iq_stStandardModuleItf.q_etDiag			:= GD.ET_Diag.Ok;
iq_stStandardModuleItf.q_udiDiagExt		:= ET_DiagExt.Disabled;
iq_stStandardModuleItf.q_sDiagExt			:= FC_EtDiagExtToString(i_etDiagExt := iq_stStandardModuleItf.q_udiDiagExt);
iq_stStandardModuleItf.q_sMsg				:= '';

iq_stStandardModuleItf.q_dwModuleType		:= TPL.ET_ModuleType.NodeModule;
iq_stStandardModuleItf.q_sModuleTypeName	:= 'NodeModule';
iq_stStandardModuleItf.q_udiModuleVersion	:= 1;	
(* End of system generated code, do not change without consulting 'Schneider Electric Automation GmbH' - otherwise you risk instability!!! *)

(* System generated code, to be changed by experienced programmers *)
IF iq_stStandardModuleItf.iq_diCMD <> 0 AND NOT iq_stStandardModuleItf.i_xEnable THEN
	iq_stStandardModuleItf.iq_diCMD := 0;
END_IF
(* End of system generated code, to be changed by experienced programmers *)

(* Application specific code *)
(* ToDo: Add your application specific code here *)
;
(* End of application specific code *)
END_ACTION

ACTION SubModules_Action:
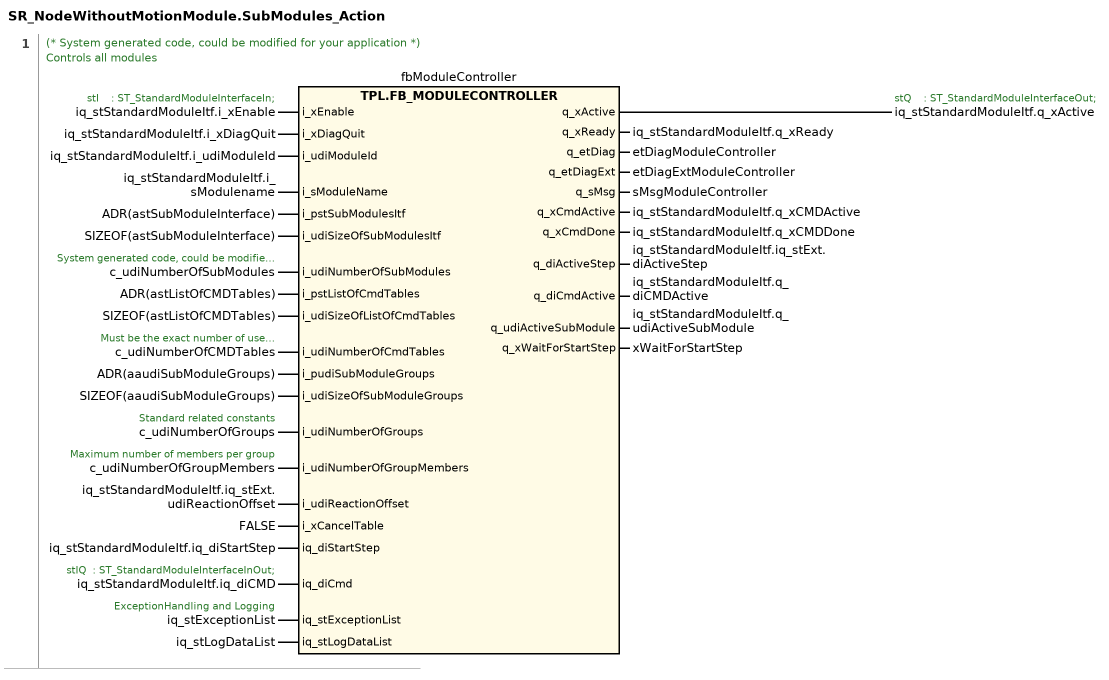
// NETWORK 1
// 					(* System generated code, could be modified for your application *)
// Controls all modules
//
//   fbModuleController: Modules related variables
//   iq_stStandardModuleItf.i_xEnable: stI : ST_StandardModuleInterfaceIn;
//   c_udiNumberOfSubModules: System generated code, could be modified for your application
//   c_udiNumberOfCMDTables: Must be the exact number of used CMDTables!
//   c_udiNumberOfGroups: Standard related constants
//   c_udiNumberOfGroupMembers: Maximum number of members per group
//   iq_stStandardModuleItf.iq_diCMD: stIQ : ST_StandardModuleInterfaceInOut;
//   iq_stExceptionList: ExceptionHandling and Logging
//   iq_stStandardModuleItf.q_xActive: stQ : ST_StandardModuleInterfaceOut;
fbModuleController(
    i_xEnable := iq_stStandardModuleItf.i_xEnable,
    i_xDiagQuit := iq_stStandardModuleItf.i_xDiagQuit,
    i_udiModuleId := iq_stStandardModuleItf.i_udiModuleId,
    i_sModuleName := iq_stStandardModuleItf.i_sModulename,
    i_pstSubModulesItf := ADR(astSubModuleInterface),
    i_udiSizeOfSubModulesItf := SIZEOF(astSubModuleInterface),
    i_udiNumberOfSubModules := c_udiNumberOfSubModules,
    i_pstListOfCmdTables := ADR(astListOfCMDTables),
    i_udiSizeOfListOfCmdTables := SIZEOF(astListOfCMDTables),
    i_udiNumberOfCmdTables := c_udiNumberOfCMDTables,
    i_pudiSubModuleGroups := ADR(aaudiSubModuleGroups),
    i_udiSizeOfSubModuleGroups := SIZEOF(aaudiSubModuleGroups),
    i_udiNumberOfGroups := c_udiNumberOfGroups,
    i_udiNumberOfGroupMembers := c_udiNumberOfGroupMembers,
    i_udiReactionOffset := iq_stStandardModuleItf.iq_stExt.udiReactionOffset,
    i_xCancelTable := FALSE,
    iq_diStartStep := iq_stStandardModuleItf.iq_diStartStep,
    iq_diCmd := iq_stStandardModuleItf.iq_diCMD,
    iq_stExceptionList := iq_stExceptionList,
    iq_stLogDataList := iq_stLogDataList,
    q_xReady => iq_stStandardModuleItf.q_xReady,
    q_etDiag => etDiagModuleController,
    q_etDiagExt => etDiagExtModuleController,
    q_sMsg => sMsgModuleController,
    q_xCmdActive => iq_stStandardModuleItf.q_xCMDActive,
    q_xCmdDone => iq_stStandardModuleItf.q_xCMDDone,
    q_diActiveStep => iq_stStandardModuleItf.iq_stExt.diActiveStep,
    q_diCmdActive => iq_stStandardModuleItf.q_diCMDActive,
    q_udiActiveSubModule => iq_stStandardModuleItf.q_udiActiveSubModule,
    q_xWaitForStartStep => xWaitForStartStep); // TPL.FB_MODULECONTROLLER
iq_stStandardModuleItf.q_xActive := fbModuleController.q_xActive;
END_ACTION

ACTION UpdateStructs:
(* System generated code, do not change without consulting 'Schneider Electric Automation GmbH' - otherwise you risk instability!!!*)
fbDetectOnlineChange(	i_xEnable	:= TRUE, 
						i_xDetect	:= TRUE, 
						q_xActive	=> xDetectOnlineChangeActive, 
						q_xReady	=> xDetectOnlineChangeReady, 
						q_etDiag	=> etDetectOnlineChangeDiag, 
						q_etDiagExt	=> etDetectOnlineChangeDiagExt, 
						q_sMsg		=> sDetectOnlineChangeMsg, 
						q_xChange	=> );
						
IF(NOT fbDetectOnlineChange.q_xChange) THEN
	RETURN;
END_IF

iq_stStandardModuleItf.iq_stExt.udiNumberOfSubModules 		:= c_udiNumberOfSubModules;
iq_stStandardModuleItf.iq_stExt.dwSubModulesItf		 		:= ADR(astSubModuleInterface);
iq_stStandardModuleItf.iq_stExt.pdwSubModulesAddItf		 	:= ADR(adwSubModuleAddInterfaces);
iq_stStandardModuleItf.iq_stExt.pstListofCMDTables			:= ADR(astListOfCMDTables);
iq_stStandardModuleItf.iq_stExt.udiNumberOfCmdTables		:= c_udiNumberOfCMDTables;
(* End of system generated code, do not change without consulting 'Schneider Electric Automation GmbH' - otherwise you risk instability!!!*)

(* System generated code, could be modified for your application *)
xUpdateStructsException := FALSE;

(*****************************************************************************************************************************************************)
(* Update CmdTable - Prepare *)

TPL.FC_UpdateCmdTableListElement(	i_pstListofCMDTables	:= ADR(astListofCMDTables),
									i_udiNumberOfCMDTables	:= c_udiNumberOfCMDTables,
									i_diCMD					:= ET_Cmd.Prepare,
									i_pstCMDTable			:= ADR(astPrepareTable),
									q_etDiag				=> etDiag,
									q_etDiagExt				=> etDiagExtTPL);
									
IF etDiag <> GD.ET_Diag.Ok AND NOT xUpdateStructsException THEN
	xUpdateStructsException := TRUE;
	
	stUpdateStructsException.sMsg := PDL.FC_MultiConcat(i_sString1 := 'Update CmdTable: Prepare - ', 
														i_sString2 := GD.FC_EtDiagToString(i_etDiag := etDiag), 
														i_sString3 := ' - ', 
														i_sString4 := TPL.FC_EtDiagExtToString(i_etDiagExt := etDiagExtTPL));
END_IF										

(*****************************************************************************************************************************************************)
(* Update CmdTable - Auto *)

TPL.FC_UpdateCmdTableListElement(	i_pstListofCMDTables	:= ADR(astListofCMDTables),
									i_udiNumberOfCMDTables	:= c_udiNumberOfCMDTables,
									i_diCMD					:= ET_Cmd.Auto,
									i_pstCMDTable			:= ADR(astAutoTable),
									q_etDiag				=> etDiag,
									q_etDiagExt				=> etDiagExtTPL);
									
IF etDiag <> GD.ET_Diag.Ok AND NOT xUpdateStructsException THEN
	xUpdateStructsException := TRUE;
	
	stUpdateStructsException.sMsg := PDL.FC_MultiConcat(i_sString1 := 'Update CmdTable: Auto - ', 
														i_sString2 := GD.FC_EtDiagToString(i_etDiag := etDiag), 
														i_sString3 := ' - ', 
														i_sString4 := TPL.FC_EtDiagExtToString(i_etDiagExt := etDiagExtTPL));
END_IF		

(*****************************************************************************************************************************************************)
(* Update CmdTable - Manual *)

TPL.FC_UpdateCmdTableListElement(	i_pstListofCMDTables	:= ADR(astListofCMDTables),
									i_udiNumberOfCMDTables	:= c_udiNumberOfCMDTables,
									i_diCMD					:= ET_Cmd.Manual,
									i_pstCMDTable			:= ADR(astManualTable),
									q_etDiag				=> etDiag,
									q_etDiagExt				=> etDiagExtTPL);
									
IF etDiag <> GD.ET_Diag.Ok AND NOT xUpdateStructsException THEN
	xUpdateStructsException := TRUE;
	
	stUpdateStructsException.sMsg := PDL.FC_MultiConcat(i_sString1 := 'Update CmdTable: Manual - ', 
														i_sString2 := GD.FC_EtDiagToString(i_etDiag := etDiag), 
														i_sString3 := ' - ', 
														i_sString4 := TPL.FC_EtDiagExtToString(i_etDiagExt := etDiagExtTPL));
END_IF		

(*****************************************************************************************************************************************************)
(* Update CmdTable - Stop *)

TPL.FC_UpdateCmdTableListElement(	i_pstListofCMDTables	:= ADR(astListofCMDTables),
									i_udiNumberOfCMDTables	:= c_udiNumberOfCMDTables,
									i_diCMD					:= ET_Cmd.Stop,
									i_pstCMDTable			:= ADR(astStopTable),
									q_etDiag				=> etDiag,
									q_etDiagExt				=> etDiagExtTPL);
									
IF etDiag <> GD.ET_Diag.Ok AND NOT xUpdateStructsException THEN
	xUpdateStructsException := TRUE;
	
	stUpdateStructsException.sMsg := PDL.FC_MultiConcat(i_sString1 := 'Update CmdTable: Stop - ', 
														i_sString2 := GD.FC_EtDiagToString(i_etDiag := etDiag), 
														i_sString3 := ' - ', 
														i_sString4 := TPL.FC_EtDiagExtToString(i_etDiagExt := etDiagExtTPL));
END_IF		

(*****************************************************************************************************************************************************)
(* Update CmdTable - Start *)

TPL.FC_UpdateCmdTableListElement(	i_pstListofCMDTables	:= ADR(astListofCMDTables),
									i_udiNumberOfCMDTables	:= c_udiNumberOfCMDTables,
									i_diCMD					:= ET_Cmd.Start,
									i_pstCMDTable			:= ADR(astStartTable),
									q_etDiag				=> etDiag,
									q_etDiagExt				=> etDiagExtTPL);
									
IF etDiag <> GD.ET_Diag.Ok AND NOT xUpdateStructsException THEN
	xUpdateStructsException := TRUE;
	
	stUpdateStructsException.sMsg := PDL.FC_MultiConcat(i_sString1 := 'Update CmdTable: Start - ', 
														i_sString2 := GD.FC_EtDiagToString(i_etDiag := etDiag), 
														i_sString3 := ' - ', 
														i_sString4 := TPL.FC_EtDiagExtToString(i_etDiagExt := etDiagExtTPL));
END_IF		

(*****************************************************************************************************************************************************)
(* Update CmdTable - Abort *)

TPL.FC_UpdateCmdTableListElement(	i_pstListofCMDTables	:= ADR(astListofCMDTables),
									i_udiNumberOfCMDTables	:= c_udiNumberOfCMDTables,
									i_diCMD					:= ET_Cmd.Abort,
									i_pstCMDTable			:= ADR(astAbortTable),
									q_etDiag				=> etDiag,
									q_etDiagExt				=> etDiagExtTPL);
									
IF etDiag <> GD.ET_Diag.Ok AND NOT xUpdateStructsException THEN
	xUpdateStructsException := TRUE;
	
	stUpdateStructsException.sMsg := PDL.FC_MultiConcat(i_sString1 := 'Update CmdTable: Abort - ', 
														i_sString2 := GD.FC_EtDiagToString(i_etDiag := etDiag), 
														i_sString3 := ' - ', 
														i_sString4 := TPL.FC_EtDiagExtToString(i_etDiagExt := etDiagExtTPL));
END_IF		

(*****************************************************************************************************************************************************)
(* Update CmdTable - Hold *)

TPL.FC_UpdateCmdTableListElement(	i_pstListofCMDTables	:= ADR(astListofCMDTables),
									i_udiNumberOfCMDTables	:= c_udiNumberOfCMDTables,
									i_diCMD					:= ET_Cmd.Hold,
									i_pstCMDTable			:= ADR(astHoldTable),
									q_etDiag				=> etDiag,
									q_etDiagExt				=> etDiagExtTPL);
									
IF etDiag <> GD.ET_Diag.Ok AND NOT xUpdateStructsException THEN
	xUpdateStructsException := TRUE;
	
	stUpdateStructsException.sMsg := PDL.FC_MultiConcat(i_sString1 := 'Update CmdTable: Hold - ', 
														i_sString2 := GD.FC_EtDiagToString(i_etDiag := etDiag), 
														i_sString3 := ' - ', 
														i_sString4 := TPL.FC_EtDiagExtToString(i_etDiagExt := etDiagExtTPL));
END_IF		

(*****************************************************************************************************************************************************)
(* Update CmdTable - BrakeRelease *)

TPL.FC_UpdateCmdTableListElement(	i_pstListofCMDTables	:= ADR(astListofCMDTables),
									i_udiNumberOfCMDTables	:= c_udiNumberOfCMDTables,
									i_diCMD					:= ET_Cmd.BrakeRelease,
									i_pstCMDTable			:= ADR(astBrakeReleaseTable),
									q_etDiag				=> etDiag,
									q_etDiagExt				=> etDiagExtTPL);
									
IF etDiag <> GD.ET_Diag.Ok AND NOT xUpdateStructsException THEN
	xUpdateStructsException := TRUE;
	
	stUpdateStructsException.sMsg := PDL.FC_MultiConcat(i_sString1 := 'Update CmdTable: BrakeRelease - ', 
														i_sString2 := GD.FC_EtDiagToString(i_etDiag := etDiag), 
														i_sString3 := ' - ', 
														i_sString4 := TPL.FC_EtDiagExtToString(i_etDiagExt := etDiagExtTPL));
END_IF		

(*****************************************************************************************************************************************************)
(* Set exception if any exception occurred *)

TPL.FC_SetException(i_xExceptionActive	:= xUpdateStructsException, 
					iq_stException		:= stUpdateStructsException, 
					iq_stExceptionList	:= iq_stExceptionList, 
					iq_stLogDataList	:= iq_stLogDataList);
					
xInitSuccessful := xInitSuccessful AND NOT xUpdateStructsException;

etDiag := GD.ET_Diag.Ok;
(* End of system generated code, could be modified for your application *)
END_ACTION

END_PROGRAM

// LMC_PacDrive/Application/FB_ExampleTableDiagSource
FUNCTION_BLOCK FB_ExampleTableDiagSource
VAR_INPUT
	i_xEnable			: BOOL;
	i_xDiagQuit			: BOOL;
END_VAR

VAR_IN_OUT
	iq_stComStructure	: TPL.ST_DiagnosticsManagerToDiagSource;
END_VAR

VAR_OUTPUT
	q_xActive			: BOOL;
	q_xReady			: BOOL;
	q_etDiag			: GD.ET_Diag := GD.ET_Diag.Ok;
	q_etDiagExt			: ET_DiagExt := ET_DiagExt.Disabled;
	q_sMsg				: STRING[80];
END_VAR

VAR
	xEnableFlag		: BOOL;
	diState			: DINT;
	
	udiOwnSourceId : UDINT := 0;

	diOldCmd	: DINT := 0;
	diCmdExecState : DINT := 0;
	
	fbTableWriter : TPL.FB_TableWriter;

	udiCName : UDINT;
	udiCValue : UDINT;
	udiCC3 : UDINT;

	udiRowCounter : UDINT := 1;
	
	etDiag			: GD.ET_Diag;
	etDiagExtTPL	: TPL.ET_DiagExt;
	sMsg			: STRING[80];
	
	rtrigDiagQuit	: Standard.R_TRIG;
END_VAR

VAR CONSTANT
	c_sName : STRING[TPL.Gc_udiTableWriterMaxNameLength] := 'I_am_something';
	c_sTypeName : STRING[TPL.Gc_udiTableWriterMaxNameLength] := 'ExampleTableDiagSource';
	c_udiMaxNumRows : UDINT := 40;
END_VAR

IF i_xEnable AND NOT xEnableFlag THEN
	xEnableFlag := TRUE;
	
	q_xActive := TRUE;
	
	SetDiagOutputs(	i_etDiag	:= GD.ET_Diag.Ok,
					i_etDiagExt	:= ET_DiagExt.WaitUntilDiagnosticsManagerReady,
					i_sMsg		:= '');	
	diState := 10;
	
ELSIF NOT i_xEnable AND xEnableFlag THEN
	xEnableFlag := FALSE;
		
	IF udiOwnSourceId <> 0 THEN		
		SetDiagOutputs(	i_etDiag	:= GD.ET_Diag.Ok,
						i_etDiagExt	:= ET_DiagExt.WaitUntilDisabled,
						i_sMsg		:= '');
		diState := 100;
		
	ELSIF udiOwnSourceId = 0 THEN		
		SetDiagOutputs(	i_etDiag	:= GD.ET_Diag.Ok,
						i_etDiagExt	:= ET_DiagExt.Disabled,
						i_sMsg		:= '');
	END_IF
END_IF

DiagQuit();

CASE diState OF
	
	0:	(* Disable & exception state *)
	
	10:	(* Wait until diagnostics manager ready *)
		IF iq_stComStructure.i_xDiagnosticsManagerReady THEN
			
			SetDiagOutputs(	i_etDiag	:= GD.ET_Diag.Ok,
							i_etDiagExt	:= ET_DiagExt.WaitUntilDiagSourceRegistered,
							i_sMsg		:= '');
			diState := 20;
		END_IF

	20:	(* Wait until diag source registered *)	
		IF NOT iq_stComStructure.i_xDiagnosticsManagerReady THEN
			
			SetDiagOutputs(	i_etDiag	:= GD.ET_Diag.Ok,
							i_etDiagExt	:= ET_DiagExt.WaitUntilDiagnosticsManagerReady,
							i_sMsg		:= '');	
			diState := 10;
			RETURN;
	
		(* only write to register structure if no one else has done it in this cylce *)
		ELSIF (NOT iq_stComStructure.iq_stRegister.xUsed AND iq_stComStructure.iq_stRegister.udiNextId <> 0) THEN
			(* register *)
			iq_stComStructure.iq_stRegister.xUsed := TRUE;
			
			iq_stComStructure.iq_stRegister.sName		:= c_sName;
			iq_stComStructure.iq_stRegister.sTypeName	:= c_sTypeName;
			
			udiOwnSourceId := iq_stComStructure.iq_stRegister.udiNextId; (* register with this id; required for the following communication *)
		ELSE
			RETURN;
		END_IF
		
		q_xReady := TRUE;
		
		SetDiagOutputs(	i_etDiag	:= GD.ET_Diag.Ok,
						i_etDiagExt	:= ET_DiagExt.WaitForCommunication,
						i_sMsg		:= '');
		diState := 30;
	
	30:	(* Wait for communication *)	
		IF NOT iq_stComStructure.i_xDiagnosticsManagerReady THEN

			CancelWriting();
									
			udiOwnSourceId	:= 0;
			
			SetDiagOutputs(	i_etDiag	:= GD.ET_Diag.Ok,
							i_etDiagExt	:= ET_DiagExt.WaitUntilDiagnosticsManagerReady,
							i_sMsg		:= '');	
			diState := 10;
			RETURN;
			
		ELSIF (iq_stComStructure.i_udiComWithId = udiOwnSourceId) THEN		(* Am I adressed? *)
			
			WriteDiagDataControl();

		ELSE
			iq_stComStructure.q_lrProgress := 0.0;
			
			CancelWriting();
						
			SetDiagOutputs(	i_etDiag	:= GD.ET_Diag.Ok,
							i_etDiagExt	:= ET_DiagExt.WaitForCommunication,
							i_sMsg		:= '');
		END_IF
		
	100: (* Wait until disabled *)	
		IF NOT iq_stComStructure.i_xDiagnosticsManagerReady THEN

			CancelWriting();
									
			udiOwnSourceId	:= 0;
			
			SetDiagOutputs(	i_etDiag	:= GD.ET_Diag.Ok,
							i_etDiagExt	:= ET_DiagExt.Disabled,
							i_sMsg		:= '');	
	
		ELSIF (iq_stComStructure.i_udiComWithId = udiOwnSourceId) THEN		(* Am I adressed? *)
			
			WriteDiagDataControl();
			
		(* only write to register structure if no one else has done it in this cylce *)
		ELSIF (NOT iq_stComStructure.iq_stRegister.xUsed AND NOT iq_stComStructure.iq_stRegister.xUnsubscribe) AND 
			   NOT iq_stComStructure.i_xDiagnosticsActive THEN
			   
			iq_stComStructure.iq_stRegister.xUsed			:= TRUE;
			
			iq_stComStructure.iq_stRegister.xUnsubscribe	:= TRUE;
			iq_stComStructure.iq_stRegister.udiSourceId		:= udiOwnSourceId;
			
			q_xActive := FALSE;
			
			SetDiagOutputs(	i_etDiag	:= GD.ET_Diag.Ok,
							i_etDiagExt	:= ET_DiagExt.Disabled,
							i_sMsg		:= '');
		END_IF
END_CASE

IF q_xActive THEN	
	IF(diCmdExecState <> 0) THEN
		WriteDiagDataToFile();
		
		IF(iq_stComStructure.iq_diCmd <= 0) THEN
			diOldCmd := iq_stComStructure.iq_diCmd;
		END_IF
	END_IF	
END_IF

{attribute 'hide'}
METHOD CancelWriting : BOOL
VAR_INPUT
END_VAR
(* Deactivate writing if we are (for whatever reason) no longer adressed.
   May happen in case network connection with Diagnostics is disrupted or Source will be disabled *)

THIS^.diOldCmd			:= 0;
THIS^.diCmdExecState	:= 0;
END_METHOD

{attribute 'hide'}
METHOD ExceptionDuringWriting : BOOL
VAR_INPUT
END_VAR
(* exception during writing *)
CASE THIS^.etDiagExtTPL OF
	TPL.ET_DiagExt.HeaderStartAlreadySuccessfullyCalled,	// FB_TableWriter.HeaderStart	
	TPL.ET_DiagExt.FileIdNotSet,							// FB_TableWriter.HeaderStart							
	TPL.ET_DiagExt.FileIdInvalid,							// FB_TableWriter.HeaderStart & FB_TableWriter.HeaderAddColumn & FB_TableWriter.HeaderFinish & FB_TableWriter.RowStart & FB_TableWriter.RowValue & FB_TableWriter.TableEnd							
	TPL.ET_DiagExt.FileNotOpen,								// FB_TableWriter.HeaderStart & FB_TableWriter.HeaderAddColumn & FB_TableWriter.HeaderFinish & FB_TableWriter.RowStart & FB_TableWriter.RowValue & FB_TableWriter.TableEnd								
	TPL.ET_DiagExt.UnexpectedFeedback,						// FB_TableWriter.HeaderStart & FB_TableWriter.HeaderAddColumn & FB_TableWriter.HeaderFinish & FB_TableWriter.RowStart & FB_TableWriter.RowValue & FB_TableWriter.TableEnd								
	TPL.ET_DiagExt.HeaderStartNotCalled,					// FB_TableWriter.HeaderAddColumn								
	TPL.ET_DiagExt.HeaderStartNotSuccessfullyCalled,		// FB_TableWriter.HeaderAddColumn								
	TPL.ET_DiagExt.MaxNumberOfColumnsExceeded,				// FB_TableWriter.HeaderAddColumn						
	TPL.ET_DiagExt.NameInvalid,								// FB_TableWriter.HeaderAddColumn								
	TPL.ET_DiagExt.NoColumnsDefined,						// FB_TableWriter.HeaderFinish	
	TPL.ET_DiagExt.DefineHeaderFirst,						// FB_TableWriter.RowStart
	TPL.ET_DiagExt.RowStartedCallRowEndFirst,				// FB_TableWriter.RowStart
	TPL.ET_DiagExt.CallRowStartFirst,						// FB_TableWriter.RowValue
	TPL.ET_DiagExt.ColumnNumberRange,						// FB_TableWriter.RowValue
	TPL.ET_DiagExt.RowsStillOpen,							// FB_TableWriter.TableEnd
	TPL.ET_DiagExt.HeaderColumnIdInvalid:
	
		SetDiagOutputs(	i_etDiag	:= GD.ET_Diag.UnexpectedProgramBehavior,
						i_etDiagExt	:= ET_DiagExt.UnexpectedFeedback,
						i_sMsg		:= PDL.FC_MultiConcat(	i_sString1	:= 'FB_TableWriter: ', 
															i_sString2	:= GD.FC_EtDiagToString(THIS^.etDiag), 
															i_sString3	:= ' - ', 
															i_sString4	:= TPL.FC_EtDiagExtToString(THIS^.etDiagExtTPL), 
															q_etDiag	=> , 
															q_etDiagExt	=> )); 								
	ELSE
		SetDiagOutputs(	i_etDiag	:= GD.ET_Diag.UnexpectedProgramBehavior,
						i_etDiagExt	:= ET_DiagExt.UnexpectedFeedback,
						i_sMsg		:= PDL.FC_MultiConcat(	i_sString1	:= 'FB_TableWriter: ', 
															i_sString2	:= GD.FC_EtDiagToString(THIS^.etDiag), 
															i_sString3	:= ' - ', 
															i_sString4	:= TPL.FC_EtDiagExtToString(THIS^.etDiagExtTPL), 
															q_etDiag	=> , 
															q_etDiagExt	=> )); 						
END_CASE
		
CancelWriting();
END_METHOD

{attribute 'hide'}
METHOD SetDiagOutputs : BOOL
VAR_INPUT
	i_etDiag		: GD.ET_Diag;
	i_etDiagExt		: ET_DiagExt;
	i_sMsg			: STRING[80];
END_VAR
IF THIS^.q_etDiag = GD.ET_Diag.Ok OR i_etDiagExt = ET_DiagExt.Disabled THEN

	IF i_etDiag <> GD.ET_Diag.Ok OR i_etDiagExt = ET_DiagExt.Disabled THEN
		
		IF i_etDiag <> GD.ET_Diag.Ok THEN
			THIS^.iq_stComStructure.iq_diCmd := -THIS^.iq_stComStructure.iq_diCmd;
		END_IF
		
		IF i_etDiagExt = ET_DiagExt.Disabled THEN
			THIS^.q_xActive := FALSE;
			
			CancelWriting();
		END_IF
		
		THIS^.q_xReady := FALSE;
		THIS^.diState := 0;
	END_IF
	
	THIS^.q_etDiag		:= i_etDiag;
	THIS^.q_etDiagExt	:= i_etDiagExt;
	THIS^.q_sMsg		:= i_sMsg;

END_IF
END_METHOD

END_FUNCTION_BLOCK

// LMC_PacDrive/Application/FB_ExampleTreeDiagSource
FUNCTION_BLOCK FB_ExampleTreeDiagSource
VAR_INPUT
	i_xEnable			: BOOL;
	i_xDiagQuit			: BOOL;
END_VAR

VAR_IN_OUT
	iq_stComStructure	: TPL.ST_DiagnosticsManagerToDiagSource;
END_VAR

VAR_OUTPUT
	q_xActive			: BOOL;
	q_xReady			: BOOL;
	q_etDiag			: GD.ET_Diag := GD.ET_Diag.Ok;
	q_etDiagExt			: ET_DiagExt := ET_DiagExt.Disabled;
	q_sMsg				: STRING[80];
END_VAR

VAR
	xEnableFlag		: BOOL;
	diState			: DINT;
	
	udiOwnSourceId : UDINT := 0;
	
	fbTreeWriter	: TPL.FB_TreeWriter;

	diOldCmd	: DINT := 0;
	diCmdExecState : DINT := 0;

	uiMaxNodePerLevel : UINT := 7;

	uiLevelCounter : UINT := 1;
	auiNodeCounter : ARRAY[1..c_uiMaxLevel] OF UINT;
	uiNodeId : UINT := 1;
	lrSumNodes : LREAL := 1;

	uiTmp : UINT := 0;
	
	etDiag			: GD.ET_Diag;
	etDiagExtTPL	: TPL.ET_DiagExt;
	sMsg			: STRING[80];
	
	rtrigDiagQuit	: Standard.R_TRIG;
END_VAR

VAR CONSTANT
	c_sName : STRING[TPL.Gc_udiTableWriterMaxNameLength] := 'I_am_a_Tree';
	c_sTypeName : STRING[TPL.Gc_udiTableWriterMaxNameLength] := 'ExampleTreeDiagSource';
	c_uiMaxLevel : UINT := 5;
END_VAR

IF i_xEnable AND NOT xEnableFlag THEN
	xEnableFlag := TRUE;
	
	q_xActive := TRUE;
	
	SetDiagOutputs(	i_etDiag	:= GD.ET_Diag.Ok,
					i_etDiagExt	:= ET_DiagExt.WaitUntilDiagnosticsManagerReady,
					i_sMsg		:= '');	
	diState := 10;
	
ELSIF NOT i_xEnable AND xEnableFlag THEN
	xEnableFlag := FALSE;
		
	IF udiOwnSourceId <> 0 THEN		
		SetDiagOutputs(	i_etDiag	:= GD.ET_Diag.Ok,
						i_etDiagExt	:= ET_DiagExt.WaitUntilDisabled,
						i_sMsg		:= '');
		diState := 100;
		
	ELSIF udiOwnSourceId = 0 THEN		
		SetDiagOutputs(	i_etDiag	:= GD.ET_Diag.Ok,
						i_etDiagExt	:= ET_DiagExt.Disabled,
						i_sMsg		:= '');
	END_IF
END_IF

DiagQuit();

CASE diState OF
	
	0:	(* Disable & exception state *)
	
	10:	(* Wait until diagnostics manager ready *)
		IF iq_stComStructure.i_xDiagnosticsManagerReady THEN
			
			SetDiagOutputs(	i_etDiag	:= GD.ET_Diag.Ok,
							i_etDiagExt	:= ET_DiagExt.WaitUntilDiagSourceRegistered,
							i_sMsg		:= '');
			diState := 20;
		END_IF

	20:	(* Wait until diag source registered *)	
		IF NOT iq_stComStructure.i_xDiagnosticsManagerReady THEN
			
			SetDiagOutputs(	i_etDiag	:= GD.ET_Diag.Ok,
							i_etDiagExt	:= ET_DiagExt.WaitUntilDiagnosticsManagerReady,
							i_sMsg		:= '');	
			diState := 10;
			RETURN;
	
		(* only write to register structure if no one else has done it in this cylce *)
		ELSIF (NOT iq_stComStructure.iq_stRegister.xUsed AND iq_stComStructure.iq_stRegister.udiNextId <> 0) THEN
			(* register *)
			iq_stComStructure.iq_stRegister.xUsed := TRUE;
			
			iq_stComStructure.iq_stRegister.sName		:= c_sName;
			iq_stComStructure.iq_stRegister.sTypeName	:= c_sTypeName;
			
			udiOwnSourceId := iq_stComStructure.iq_stRegister.udiNextId; (* register with this id; required for the following communication *)
		ELSE
			RETURN;
		END_IF
		
		q_xReady := TRUE;
		
		SetDiagOutputs(	i_etDiag	:= GD.ET_Diag.Ok,
						i_etDiagExt	:= ET_DiagExt.WaitForCommunication,
						i_sMsg		:= '');
		diState := 30;
	
	30:	(* Wait for communication *)	
		IF NOT iq_stComStructure.i_xDiagnosticsManagerReady THEN

			CancelWriting();
									
			udiOwnSourceId	:= 0;
			
			SetDiagOutputs(	i_etDiag	:= GD.ET_Diag.Ok,
							i_etDiagExt	:= ET_DiagExt.WaitUntilDiagnosticsManagerReady,
							i_sMsg		:= '');	
			diState := 10;
			RETURN;
			
		ELSIF (iq_stComStructure.i_udiComWithId = udiOwnSourceId) THEN		(* Am I adressed? *)
			
			WriteDiagDataControl();

		ELSE
			iq_stComStructure.q_lrProgress := 0.0;
			
			CancelWriting();
						
			SetDiagOutputs(	i_etDiag	:= GD.ET_Diag.Ok,
							i_etDiagExt	:= ET_DiagExt.WaitForCommunication,
							i_sMsg		:= '');
		END_IF
		
	100: (* Wait until disabled *)	
		IF NOT iq_stComStructure.i_xDiagnosticsManagerReady THEN

			CancelWriting();
									
			udiOwnSourceId	:= 0;
			
			SetDiagOutputs(	i_etDiag	:= GD.ET_Diag.Ok,
							i_etDiagExt	:= ET_DiagExt.Disabled,
							i_sMsg		:= '');	
	
		ELSIF (iq_stComStructure.i_udiComWithId = udiOwnSourceId) THEN		(* Am I adressed? *)
			
			WriteDiagDataControl();
			
		(* only write to register structure if no one else has done it in this cylce *)
		ELSIF (NOT iq_stComStructure.iq_stRegister.xUsed AND NOT iq_stComStructure.iq_stRegister.xUnsubscribe) AND 
			   NOT iq_stComStructure.i_xDiagnosticsActive THEN
			   
			iq_stComStructure.iq_stRegister.xUsed			:= TRUE;
			
			iq_stComStructure.iq_stRegister.xUnsubscribe	:= TRUE;
			iq_stComStructure.iq_stRegister.udiSourceId		:= udiOwnSourceId;
			
			q_xActive := FALSE;
			
			SetDiagOutputs(	i_etDiag	:= GD.ET_Diag.Ok,
							i_etDiagExt	:= ET_DiagExt.Disabled,
							i_sMsg		:= '');
		END_IF
END_CASE

IF q_xActive THEN	
	IF(diCmdExecState <> 0) THEN
		WriteDiagDataToFile();
		
		IF(iq_stComStructure.iq_diCmd <= 0) THEN
			diOldCmd := iq_stComStructure.iq_diCmd;
		END_IF
	END_IF	
END_IF

{attribute 'hide'}
METHOD CancelWriting : BOOL
VAR_INPUT
END_VAR
(* Deactivate writing if we are (for whatever reason) no longer adressed.
   May happen in case network connection with Diagnostics is disrupted or Source will be disabled *)

THIS^.diOldCmd			:= 0;
THIS^.diCmdExecState	:= 0;
END_METHOD

{attribute 'hide'}
METHOD ExceptionDuringWriting : BOOL
VAR_INPUT
END_VAR
(* exception during writing *)
CASE THIS^.etDiagExtTPL OF
	TPL.ET_DiagExt.TreeStartAlreadySuccessfullyCalled,		// FB_TreeWriter.TreeStart	
	TPL.ET_DiagExt.FileIdNotSet,							// FB_TreeWriter.TreeStart							
	TPL.ET_DiagExt.FileIdInvalid,							// FB_TreeWriter.TreeStart & FB_TreeWriter.NodeStart & FB_TreeWriter.Parameter & FB_TreeWriter.NodeEnd & FB_TreeWriter.TreeEnd								
	TPL.ET_DiagExt.FileNotOpen,								// FB_TreeWriter.TreeStart & FB_TreeWriter.NodeStart & FB_TreeWriter.Parameter & FB_TreeWriter.NodeEnd & FB_TreeWriter.TreeEnd								
	TPL.ET_DiagExt.UnexpectedFeedback,						// FB_TreeWriter.TreeStart & FB_TreeWriter.NodeStart & FB_TreeWriter.Parameter & FB_TreeWriter.NodeEnd & FB_TreeWriter.TreeEnd								
	TPL.ET_DiagExt.TreeStartNotCalled,						// FB_TreeWriter.NodeStart								
	TPL.ET_DiagExt.TreeStartNotSuccessfullyCalled,			// FB_TreeWriter.NodeStart								
	TPL.ET_DiagExt.NoMoreNodeOpen,							// FB_TreeWriter.Parameter & FB_TreeWriter.NodeEnd						
	TPL.ET_DiagExt.CallTreeStartFirst,						// FB_TreeWriter.TreeEnd								
	TPL.ET_DiagExt.NodesStillOpen:							// FB_TreeWriter.TreeEnd	
	
		SetDiagOutputs(	i_etDiag	:= GD.ET_Diag.UnexpectedProgramBehavior,
						i_etDiagExt	:= ET_DiagExt.UnexpectedFeedback,
						i_sMsg		:= PDL.FC_MultiConcat(	i_sString1	:= 'FB_TreeWriter: ', 
															i_sString2	:= GD.FC_EtDiagToString(THIS^.etDiag), 
															i_sString3	:= ' - ', 
															i_sString4	:= TPL.FC_EtDiagExtToString(THIS^.etDiagExtTPL), 
															q_etDiag	=> , 
															q_etDiagExt	=> )); 								
	ELSE
		SetDiagOutputs(	i_etDiag	:= GD.ET_Diag.UnexpectedProgramBehavior,
						i_etDiagExt	:= ET_DiagExt.UnexpectedFeedback,
						i_sMsg		:= PDL.FC_MultiConcat(	i_sString1	:= 'FB_TreeWriter: ', 
															i_sString2	:= GD.FC_EtDiagToString(THIS^.etDiag), 
															i_sString3	:= ' - ', 
															i_sString4	:= TPL.FC_EtDiagExtToString(THIS^.etDiagExtTPL), 
															q_etDiag	=> , 
															q_etDiagExt	=> )); 						
END_CASE
		
CancelWriting();
END_METHOD

{attribute 'hide'}
METHOD SetDiagOutputs : BOOL
VAR_INPUT
	i_etDiag		: GD.ET_Diag;
	i_etDiagExt		: ET_DiagExt;
	i_sMsg			: STRING[80];
END_VAR
IF THIS^.q_etDiag = GD.ET_Diag.Ok OR i_etDiagExt = ET_DiagExt.Disabled THEN

	IF i_etDiag <> GD.ET_Diag.Ok OR i_etDiagExt = ET_DiagExt.Disabled THEN
		
		IF i_etDiag <> GD.ET_Diag.Ok THEN
			THIS^.iq_stComStructure.iq_diCmd := -THIS^.iq_stComStructure.iq_diCmd;
		END_IF
		
		IF i_etDiagExt = ET_DiagExt.Disabled THEN
			THIS^.q_xActive := FALSE;
			
			CancelWriting();
		END_IF
		
		THIS^.q_xReady := FALSE;
		THIS^.diState := 0;
	END_IF
	
	THIS^.q_etDiag		:= i_etDiag;
	THIS^.q_etDiagExt	:= i_etDiagExt;
	THIS^.q_sMsg		:= i_sMsg;

END_IF
END_METHOD

END_FUNCTION_BLOCK

// LMC_PacDrive/Application/CrankModuleExample/TaskCalls/SR_Logging
PROGRAM SR_Logging

VAR
	fbLogDataControl	: TPL.FB_LogDataControl;
END_VAR

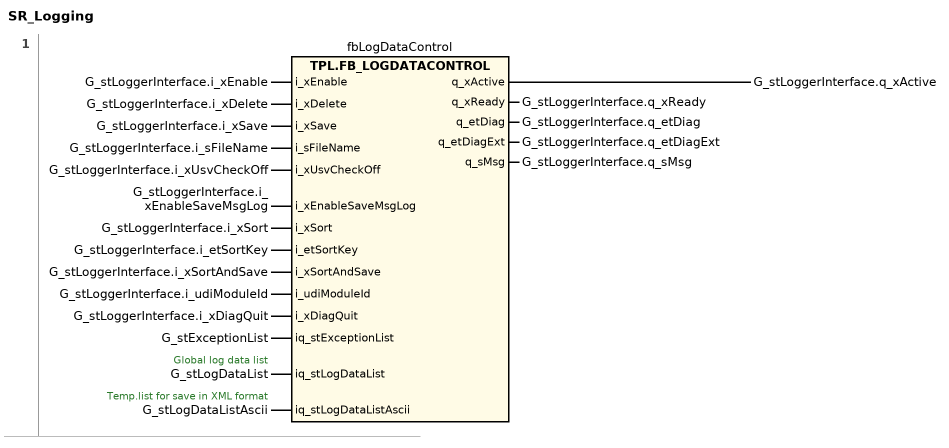
// NETWORK 1
//   G_stLogDataList: Global log data list
//   G_stLogDataListAscii: Temp.list for save in XML format
fbLogDataControl(
    i_xEnable := G_stLoggerInterface.i_xEnable,
    i_xDelete := G_stLoggerInterface.i_xDelete,
    i_xSave := G_stLoggerInterface.i_xSave,
    i_sFileName := G_stLoggerInterface.i_sFileName,
    i_xUsvCheckOff := G_stLoggerInterface.i_xUsvCheckOff,
    i_xEnableSaveMsgLog := G_stLoggerInterface.i_xEnableSaveMsgLog,
    i_xSort := G_stLoggerInterface.i_xSort,
    i_etSortKey := G_stLoggerInterface.i_etSortKey,
    i_xSortAndSave := G_stLoggerInterface.i_xSortAndSave,
    i_udiModuleId := G_stLoggerInterface.i_udiModuleId,
    i_xDiagQuit := G_stLoggerInterface.i_xDiagQuit,
    iq_stExceptionList := G_stExceptionList,
    iq_stLogDataList := G_stLogDataList,
    iq_stLogDataListAscii := G_stLogDataListAscii,
    q_xReady => G_stLoggerInterface.q_xReady,
    q_etDiag => G_stLoggerInterface.q_etDiag,
    q_etDiagExt => G_stLoggerInterface.q_etDiagExt,
    q_sMsg => G_stLoggerInterface.q_sMsg); // TPL.FB_LOGDATACONTROL
G_stLoggerInterface.q_xActive := fbLogDataControl.q_xActive;

END_PROGRAM

// LMC_PacDrive/Application/CrankModuleExample/TaskCalls/SR_HWCopyIO
PROGRAM SR_HWCopyIO

VAR
END_VAR

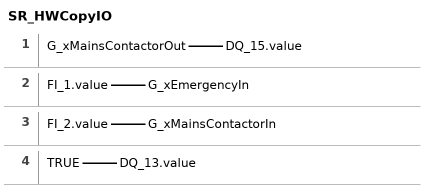
// NETWORK 1
DQ_15.value := G_xMainsContactorOut;

// NETWORK 2
G_xEmergencyIn := FI_1.value;

// NETWORK 3
G_xMainsContactorIn := FI_2.value;

// NETWORK 4
DQ_13.value := TRUE;

END_PROGRAM

// LMC_PacDrive/Application/CrankModuleExample/TaskCalls/SR_VisControl
PROGRAM SR_VisControl

VAR CONSTANT
	c_udiMaxHierarchyLevels	: UDINT := 10;
	c_stEmptyCmdTableStep	: TPL.ST_Cmd := (	sTitle			:= '',
												diStep			:= 0,
												udiModuleName	:= 0,
												diCmd			:= 0,
												timTimeOut		:= T#60S,
												xEndCmd			:= FALSE);
END_VAR

VAR (*User specific variables*)
END_VAR


VAR
	iState							: INT:= 0;
	vpq_xDoEnable 					: BOOL:= FALSE;
	xEnableFlag 					: BOOL;
	iDoEnableCycleCounter			: INT:=0;
	
	IFB_RTOPMode					: STANDARD.R_TRIG;

(* Cmd table of main machine on VIS_Main *)
	pstStep 						: POINTER TO TPL.ST_Cmd;
	udiCounter						: UDINT;
	
	vpq_astActualCmdTableMain	: ARRAY [1..10] OF TPL.ST_Cmd;
	vpq_udiNumberOfCmdStepsMain	: UDINT;
	vpq_sCmdTitelMain		: STRING;
	vpiq_udiIndexMinMain		: UDINT := 1;
	udiIndexMaxMainTable			: UDINT := 1;
	udiIndexOldMainTable			: UDINT := 1;
	
	vpq_xDisableScrollUpMain	: BOOL;
	vpq_xDisableScrollDownMain	: BOOL;

	(* Visualization of the main machine on the VIS_Main *)
	vpq_stMachineInterface				: TPL.ST_StandardModuleInterface;
	
	vpq_xMachineInException				: BOOL;	
	vpq_etMainModuleControllerDiag		: GD.ET_Diag;
	vpq_etMainModuleControllerDiagExt	: TPL.ET_DiagExt;
	vpq_sMainModuleControllerMsg			: STRING[80];

(*Exception*)
	vpiq_xTestUserException1				: BOOL;
	xTestUserException1Old					: BOOL;
	vpiq_xTestUserException2				: BOOL;
	xTestUserException2Old					: BOOL;
	vpiq_xTestUserException3				: BOOL;
	xTestUserException3Old					: BOOL;
	vpiq_xTestUserException4				: BOOL;
	xTestUserException4Old					: BOOL;
	vpiq_xTestUserException5				: BOOL;
	xTestUserException5Old					: BOOL;

	vpq_udiReactionIndexMin				: UDINT := 1;
	udiReactionIndexMax				: UDINT := 1;
	udiReactionIndexOld				: UDINT := 1;
	vpq_axReaction						: ARRAY[1..10] OF BOOL;
	
	udiCount						: UDINT;
	stActiveReactions				: TPL.ST_Reaction;
	vpiq_xReactionUp						: BOOL;
	vpiq_xReactionDown					: BOOL;

(*Vis*)
	vpiq_xShowControlFrame			: BOOL;
	vpiq_xShowModuleInterface		: BOOL;
	vpiq_iPositionX					: INT;
	vpiq_iPositionY					: INT;

	vpq_xShowLogDataListDetails				: BOOL := FALSE;
	vpiq_xButtonLogDataListDetails			: BOOL := FALSE;

	(* Visualization of the actCmdTable of the current module *)
	pstEQCMDTable							: POINTER TO TPL.ST_Cmd;		(* Pointer to active CMD Table *)
	pstEQCMDTableEntry						: POINTER TO TPL.ST_Cmd;
	vpq_astActualCmdTableModule				: ARRAY[1..10] OF TPL.ST_Cmd;
	vpiq_udiIndexMinModule						: UDINT := 1;
	udiEQTableIndexMax						: UDINT := 1;
	udiEQTableIndexOld						: UDINT := 1;
	vpq_udiNumberOfCmdStepsModule			: UDINT := 0;
	pstEQCMDTableListEntry					: POINTER TO TPL.ST_CmdTable;
	vpq_sCmdTitleModule						: STRING[80];
	udiEQTableStepCountOld					: UDINT;

	(* Navigation in the command table *)
	vpq_xDisableScrollUpModule				: BOOL;
	vpq_xDisableScrollDownModule			: BOOL;
	vpq_xDisplayCmdTable					: BOOL;

	(* 2d navigation buttons *)
	vpiq_xNavUp								: BOOL;
	vpiq_xNavDown							: BOOL;
	vpiq_xNavLeft							: BOOL;
	vpiq_xNavRight							: BOOL;
	vpq_xEnableNavUp						: BOOL;
	vpq_xEnableNavDown						: BOOL;
	vpq_xEnableNavLeft						: BOOL;
	vpq_xEnableNavRight						: BOOL;
	vpq_sNameNavUp							: STRING[80];
	vpq_sNameNavDown						: STRING[80];
	vpq_sNameNavLeft						: STRING[80];
	vpq_sNameNavRight						: STRING[80];

	(* Navigation flags *)
	pstCurrentParent						: POINTER TO TPL.ST_StandardModuleInterface;
	pstCurrent								: POINTER TO TPL.ST_StandardModuleInterface;
	xCurrentIsNoNodeModule    				: BOOL;
	dwCurrentAddInterface					: DWORD;
	xUpdateForOtherFBs						: BOOL;
	audiHierarchy							: ARRAY[1..c_udiMaxHierarchyLevels] OF UDINT; (* Selected modules in each level of the hierarchy *)
	udiCurrentLevel							: UDINT := 1; (* Level of the hierarchy we are working on*)
	udiCurrentLevelSize						: UDINT := 1;
	xCurrentHasSubModules					: BOOL := FALSE;
	pstTmp									: POINTER TO TPL.ST_StandardModuleInterface;
	pdwTmp									: POINTER TO DWORD;

	xUpdateData 							: BOOL := FALSE;
	dwDummy									: DWORD;

	vpq_xButtonSetJogTargetInvisible		: BOOL := FALSE;
	vpiq_xButtonSetCurrentAsJogTarget					: BOOL;
	vpq_xCurrentIsJogTarget						: BOOL := FALSE;
	udiSetAsJogTarget						: UDINT;
//	udiSetAsJogTargetNum					: UDINT;
	IFB_FTrigxCurrentIsJogTarget			: STANDARD.F_TRIG;

	(* Direct navigation buttons *)
	axClearBoolA5							: ARRAY[1..5] OF BOOL;
	
	vpiq_xModuleListDown							: BOOL; (* Module table scroll buttons *)
	vpq_xDisableModuleListDown					: BOOL;
	vpiq_xModuleListUp							: BOOL;
	vpq_xDisableModuleListUp						: BOOL;
	vpiq_axModuleList							: ARRAY[1..5] OF BOOL;
	vpiq_axControlModuleList						: ARRAY[1..5] OF BOOL;
	vpq_axDisableModuleList						: ARRAY[1..5] OF BOOL;
	vpq_axActiveModuleList						: ARRAY[1..5] OF BOOL; (* Highlight active module *)
	vpq_axControlModuleActive						: ARRAY[1..5] OF BOOL; (* Highlight active control module *)
	vpq_audiIdModuleList							: ARRAY[1..5] OF UDINT; (* Module ids *)
	vpq_axIdModuleListValid					: ARRAY[1..5] OF BOOL;
	vpq_axControlModuleValid					: ARRAY[1..5] OF BOOL;
	audiControlModuleNumber					: ARRAY[1..5] OF UDINT;
	vpq_asNameModuleList						: ARRAY[1..5] OF STRING[80]; (* Module name *)
	vpq_asToolTipControlModuleList				: ARRAY[1..5] OF STRING[80];
	vpq_asControlModuleButtonName				: ARRAY[1..5] OF STRING[60];
	udiNumberOfControlModulesLevel2			: UDINT;

	vpiq_xSubModuleListDown					: BOOL;
	vpq_xDisableSubModuleListDown			: BOOL;
	vpiq_xSubModuleListUp					: BOOL;
	vpq_xDisableSubModuleListUp				: BOOL;
	
	vpiq_axSubModuleList							: ARRAY[1..5] OF BOOL;
	vpq_axDisableSubModuleList					: ARRAY[1..5] OF BOOL;
	vpq_axActiveSubModuleList					: ARRAY[1..5] OF BOOL; (* Highlight active module *)
	vpq_audiIdSubModuleList					: ARRAY[1..5] OF UDINT; (* Module ids *)
	vpq_axIdSubModuleListValid						: ARRAY[1..5] OF BOOL;
	vpq_asNameSubModuleList						: ARRAY[1..5] OF STRING[60]; (* Module names *)
	vpiq_axSubControlModuleList					: ARRAY[1..5] OF BOOL;
	vpq_axSubControlModuleValid					: ARRAY[1..5] OF BOOL;
	audiSubControlModuleID					: ARRAY[1..5] OF UDINT;
	vpq_asToolTipSubControlModuleList			: ARRAY[1..5] OF STRING[80];
	vpq_axSubControlModuleActive					: ARRAY[1..5] OF BOOL;
	vpq_asSubControlModuleButtonName			: ARRAY[1..5] OF STRING[60];
	udiCurrentLevel3Size					: UDINT := 0; (* How many submodules does the current module have on level 2 *)
	pstCurrentFirstLevel3Module				: POINTER TO TPL.ST_StandardModuleInterface;
	udiCurrentNumberOfControlModules 		: UDINT;

	(*Variables for selecting control modules *)
	vpq_udiActiveControlModuleNumber				: UDINT;
	pstCurrentNodeInterface						: POINTER TO TPL.ST_StandardModuleInterface;
	pstControlModuleInterface					: POINTER TO TPL.ST_ControlModuleInterface;
	pstCurrentControlModuleStandardInterface	: POINTER TO TPL.ST_ControlModuleInterface;
	pstTempCtrlModule							: POINTER TO TPL.ST_ControlModuleInterface;
	stCurrentControlModuleStandardInterface		: TPL.ST_ControlModuleInterface;
	udiControlModuleSelectedInLevel				: UDINT;
	xControlModuleSelected						: BOOL;
	xCurrentHasControlModules					: BOOL;
	pstCurrentLevel2							: POINTER TO TPL.ST_StandardModuleInterface;

	(* Direct navigation flags *)
	udiMinModuleList						: UDINT;
	udiMinSubModuleList						: UDINT;

	(* Struct for displaying values of the current module *)
	vpq_stCurrentModuleStandardInterface		: TPL.ST_StandardModuleInterface;
	vpq_sCurrentModuleReaction				: STRING[255];
	stDummyStandardInterface				: TPL.ST_StandardModuleInterface;
	
	(* Exceptions the vis can create *)
	stPointerException						: TPL.ST_Exception;
	xPointerExceptionActive					: BOOL;


	udiSetAsCurrentModule					: UDINT; (* If <> 0, specifies the ID of a module, to set as current module *)

	(* Flags of the SetCurrentModule action *)
	udiTmp2									: UDINT;
	udiTmp									: UDINT;


	(* Inputs, for module control *)
	vpiq_diCmdToSet								: DINT;
	vpiq_diStartStepToSet					: DINT;
	vpiq_xSetCmdClicked							: BOOL; (* Set by the vis, reset by SR_VisControl, if true, diCmdToSet is written to the CMD of the current module *)
	xDiagQuit_Touch						: BOOL; (* Set by the vis, if true, the DiagQuit Input of the module is set *)
	xDiagQuit_WasTouched					: BOOL;	(* Internal flag *)
	vpiq_xEnableModuleClicked					: BOOL; (* Set by the vis, reset by SR_VisControl, if true, the xEnable of the module is toggled *)

	stModuleReactions						: TPL.ST_Reaction;
	vpiq_xModuleReactionUp						: BOOL;
	vpiq_xModuleReactionDown						: BOOL;
	vpq_udiModuleReactionIndexMin				: UDINT := 1;
	udiModuleReactionIndexMax				: UDINT := 1;
	udiModuleReactionIndexOld				: UDINT := 1;
	vpq_axModuleReaction						: ARRAY[1..10] OF BOOL;
	udiCount2								: UDINT;
	udiMaxValue								: UDINT;


	(*FR_ExceptionList, navigation in the global ExceptionList*)
	vpiq_udiExceptionListIndexMin			: UDINT := 1;
	vpq_asReaction							: ARRAY[1..10] OF STRING[80];
	vpq_udiExceptionListIndexMax				: UDINT := 1;
	vpq_xDisplayScrollDown					: BOOL;
	vpq_astExceptionListTable				: ARRAY[1..10] OF TPL.ST_Exception;
	vpiq_udiExceptionListGoToDetailsOfLine	: UDINT; (* index of the line that was selected in the exception list; set by vis to value, restet by VisControl; *)

	vpq_xShowExtendedTimes 					: BOOL := FALSE;
	vpq_xShowExtended2						: BOOL := FALSE;	
	vpiq_xButtonShowExtendedTimes 			: BOOL := FALSE;
	vpiq_xButtonShowExtended2				: BOOL := FALSE;
	
	vpq_udiNumberOfExceptions				: UDINT;
	
	udiIndex								: UDINT;
	vpq_sAllActiveReactions						: STRING[255];
	(* --- exception list --- *)

	udiExceptionListDetailsSelectIndex 		: UDINT;

	(*FR_ASCIILoggerList, navigation in the LoggerList*)
	vpiq_udiLogDataListIndexMin				: UDINT := 1;
	vpq_udiLogDataListIndexMax				: UDINT := 1;
	vpiq_udiNumberOfLogData					: UDINT;
	vpq_xLogDataScrollDown					: BOOL;
	vpq_astLogDataTableAscii				: ARRAY[1..12] OF TPL.ST_LogDataAscii;
	vpq_astLogDataTable						: ARRAY[1..12] OF TPL.ST_LogData;
	udiIndex2								: UDINT;
	udiIndex3								: UDINT;

	(*Variables to change color of the DiagQuit button*)
	vpq_dwDiagQuitColor					: DWORD;
	xRedColor							: BOOL;


	(* test exceptions *)
	stUserException1						: TPL.ST_Exception;
	stUserException2						: TPL.ST_Exception;
	stUserException3						: TPL.ST_Exception;
	stUserException4						: TPL.ST_Exception;
	stUserException5						: TPL.ST_Exception;

	(* copy of the ExceptionList *)
	fbCopyExceptionList						: TPL.FB_CopyExceptionList;
	astExceptionListCopy 					: ARRAY[1..TPL.Gc_udiMaxNumberOfExceptions] OF TPL.ST_Exception;
	
	vpiq_fbVisContExHandling					: TPL.FB_VisControllerExceptionHandling;

	(* Additional FBs for other types of modules *)
	vpiq_fbAxisModuleVisController : AXM.FB_AxisModuleVisController;
	(* For the CrankModule *)
	vpiq_fbCrankModuleVisController: CRKM.FB_CrankModuleVisController;
	
	//Crank Module variables
	vpq_xFrameSetCrankLeftInvisible	: BOOL;
	vpq_xFrameCrankDataInvisible	: BOOL;


	(* For the ExampleLeafModule *)
	vpiq_fbExampleLeafModuleVisController : FB_ExampleLeafModuleVisController;


	fbDetectOnlineChange					: TPL.FB_DetectOnlineChange;
	xDetectOnlineChangeActive				: BOOL; 
	xDetectOnlineChangeReady				: BOOL; 
	etDetectOnlineChangeDiag				: GD.ET_Diag;
	etDetectOnlineChangeDiagExt				: TPL.ET_DiagExt; 
	sDetectOnlineChangeMsg					: STRING[80];
	xUpdatePointer							: BOOL;
	fbLoggerPoint							: APL.FB_LoggerPoint;
	
	(* Highlight the currently active OpMode (VIS_AxisModule) *)
	v_diLastOpMode							: DINT;
	v_xHomeModeActive						: BOOL;
	v_xManualModeActive						: BOOL;
	v_xMultiCamCSActive						: BOOL;
	v_xMultiCamWSActive						: BOOL;
	v_xEndlessActive						: BOOL;
	v_xEndlessILSActive						: BOOL;
	v_xPositioningActive					: BOOL;
	v_xBrakeActive							: BOOL;
	v_xAdditionalCSActive					: BOOL;
	v_xAdditionalWSActive					: BOOL;
END_VAR

(* Make sure that after an online-change, the main machine program has been executed
   before you update the pointers in the VisControl. *)
   
fbDetectOnlineChange(	i_xEnable	:= TRUE, 
						i_xDetect	:= TRUE, 
						q_xActive	=> xDetectOnlineChangeActive, 
						q_xReady	=> xDetectOnlineChangeReady, 
						q_etDiag	=> etDetectOnlineChangeDiag, 
						q_etDiagExt	=> etDetectOnlineChangeDiagExt, 
						q_sMsg		=> sDetectOnlineChangeMsg, 
						q_xChange	=> );
							
IF fbDetectOnlineChange.q_xChange THEN
	xUpdatePointer := TRUE;
	RETURN;
END_IF
	
	IF G_xDoEnableVis THEN
		IF SR_MainMachine.stMachineInterface.q_xActive AND (iDoEnableCycleCounter < 3) THEN
			(* Wait until main machine is active, otherwise some module vis
			controllers would read a wrong module structure. *)
			
			iDoEnableCycleCounter := iDoEnableCycleCounter + 1;
			IF iDoEnableCycleCounter >= 3 THEN
				(* This also assures, that all values and structures are initialized
				by the main machine when this task tries to access them. *)
				vpq_xDoEnable := TRUE;
			END_IF
		END_IF
		
	ELSE
		vpq_xDoEnable := FALSE;
		iDoEnableCycleCounter := 0;
	END_IF;


IF vpq_xDoEnable AND NOT xEnableFlag THEN
	xEnableFlag := TRUE;
	
	(* Initialize navigation *)
	pstCurrentParent			:= 0;
	pstCurrent					:= ADR(SR_MainMachine.stMachineInterface);
	udiCurrentLevel				:= 1;
	udiCurrentLevelSize			:= 1;
	audiHierarchy[1]			:= 1;
	xCurrentHasSubModules		:= (pstCurrent^.iq_stExt.udiNumberOfSubModules > 0);
	xCurrentHasControlModules	:= (pstCurrent^.iq_stExt.udiNumberOfControlModules > 0);
	xPointerExceptionActive		:= FALSE;
	xUpdateData					:= TRUE;
	udiMinModuleList			:= 1;
	udiMinSubModuleList			:= 1;
	udiCurrentLevel3Size		:= 0;
	vpiq_axModuleList			:= axClearBoolA5;
	vpiq_axSubModuleList			:= axClearBoolA5;

	udiCurrentNumberOfControlModules	:= 0;
	udiNumberOfControlModulesLevel2		:= 0;
	udiControlModuleSelectedInLevel		:= 0;
	vpq_udiActiveControlModuleNumber		:= 0;

	(* init test exceptions *)
	vpq_stMachineInterface := SR_MainMachine.stMachineInterface; (* required *)
	
	InitTestExceptions();

	vpq_xCurrentIsJogTarget := FALSE;
	
	fbLoggerPoint.RegisterLoggerPoint(	i_ifParent	:= APL.G_ifApplicationLogger,
										i_sName		:= 'VisControl',
										i_sType		:= 'SR_VisControl',
										i_sSource	:= 'Project',
										q_etDiag	=> ,
										q_etDiagExt	=> );
	iState := 10;
		
ELSIF NOT vpq_xDoEnable AND xEnableFlag THEN
	xEnableFlag := FALSE;
	
	G_xPrepareActive		:= FALSE;
	G_xAutoActive			:= FALSE;
	G_xManualActive			:= FALSE;
	G_xJogMachineActive		:= FALSE;
	G_xBrakeReleaseActive	:= FALSE;
	
	iState := 5;
END_IF

CASE iState OF

0:
	iState := 5;

5:
	;

10:

	OpModeControl();

	(* Copy the machine interface into local variable, the local variable is read by the vis *)
	vpq_stMachineInterface := SR_MainMachine.stMachineInterface;

	vpq_xMachineInException := G_stExceptionList.udiNumberOfActiveExceptions > 0;

	vpq_etMainModuleControllerDiag		:= SR_MainMachine.fbModuleController.q_etDiag;
	vpq_etMainModuleControllerDiagExt	:= SR_MainMachine.fbModuleController.q_etDiagExt;
	vpq_sMainModuleControllerMsg			:= SR_MainMachine.fbModuleController.q_sMsg;

	MainPageCmdTable();
	
	ExceptionVis();

	LoggerVis();
	
	CrankModuleVis();
	
	IF (G_xDiagQuitEpas AND xPointerExceptionActive) THEN
		xPointerExceptionActive := FALSE;
		
		udiCurrentLevel					:= 1;
		audiHierarchy[udiCurrentLevel]	:= 1;
		udiCurrentLevelSize				:= 1;
		xUpdateData						:= TRUE;
		vpiq_xButtonSetCurrentAsJogTarget			:= FALSE;
	END_IF

	IF (NOT xPointerExceptionActive) THEN

		ModuleNavigationIn();

		IF (xUpdateData OR xUpdatePointer) THEN
			xUpdateData		:= FALSE;
			xUpdatePointer	:= FALSE;
			
			xUpdateForOtherFBs := TRUE;

			(* Select current module *)
			SearchCurrentModule();

			ModuleNavigationOut();

		END_IF (* xUpdateData *)

		ModuleReaction();

		(* Cyclic reading of values from the structures *)
		IF pstCurrent <> 0 THEN (* Security check *)

			(* Execute user inputs first *)
			IF(vpiq_xEnableModuleClicked) THEN
				vpiq_xEnableModuleClicked := FALSE;
				pstCurrent^.i_xEnable := NOT pstCurrent^.i_xEnable;
			END_IF
			
			IF(vpiq_xSetCmdClicked) THEN
				vpiq_xSetCmdClicked := FALSE;
				pstCurrent^.iq_diCmd := vpiq_diCmdToSet;
				pstCurrent^.iq_diStartStep := vpiq_diStartStepToSet;
			END_IF
			
			IF(xDiagQuit_Touch) THEN
				xDiagQuit_WasTouched 		:= TRUE;
				pstCurrent^.i_xDiagQuit 	:= TRUE;
			ELSIF(xDiagQuit_WasTouched) THEN
				xDiagQuit_WasTouched 		:= FALSE;
				pstCurrent^.i_xDiagQuit 	:= FALSE;
			END_IF
			
			vpq_stCurrentModuleStandardInterface := pstCurrent^;


			(* If the current module is not selected as target for the jogForw, jogBack Buttons *)
			vpq_xCurrentIsJogTarget := (vpq_stCurrentModuleStandardInterface.i_udiModuleId = SR_MainMachine.stMachineMotionInterface.i_udiModuleSelect);
			
			(* this detects a change of the current module ==> the user has navigated to a different module.
				To avoid that the old and no longer visible module is jogged further, delete the jog target *)
			IFB_FTrigxCurrentIsJogTarget(CLK:= vpq_xCurrentIsJogTarget );
			IF IFB_FTrigxCurrentIsJogTarget.Q THEN
				G_udiManualModuleSelect := 0;	(*No Module can be jogged unintentionally*)
			END_IF

		ELSE
			vpq_stCurrentModuleStandardInterface	:= stDummyStandardInterface;
			udiCurrentLevelSize					:= 0;
			xCurrentHasSubModules				:= FALSE;
			udiCurrentLevel						:= 1;
			xUpdateData							:= TRUE;
			vpq_xCurrentIsJogTarget					:= FALSE;
		END_IF

		IF pstCurrentControlModuleStandardInterface <> 0 AND vpq_udiActiveControlModuleNumber > 0 THEN
			pstTempCtrlModule := pstCurrentControlModuleStandardInterface +  UDINT_TO_DWORD((vpq_udiActiveControlModuleNumber-1) * SIZEOF(pstCurrentControlModuleStandardInterface^));
			stCurrentControlModuleStandardInterface := pstTempCtrlModule^;
		ELSE
			stCurrentControlModuleStandardInterface.udiControlModuleNumber			:= 0;
			stCurrentControlModuleStandardInterface.udiControlModuleType			:= 0;
			stCurrentControlModuleStandardInterface.dwControlModuleAddItf			:= 0;
			stCurrentControlModuleStandardInterface.sControlModuleName				:= '';
		END_IF

		vpq_xButtonSetJogTargetInvisible := NOT SR_MainMachine.xOutputManualActive;

		(* Select the current module as target for the jogging *)
		IF(SR_MainMachine.xOutputManualActive) THEN
			(* Check whether we are really in jog mode *)
			IF(vpiq_xButtonSetCurrentAsJogTarget) THEN
				G_udiManualModuleSelect := vpq_stCurrentModuleStandardInterface.i_udiModuleId;
			END_IF
		END_IF
		
		vpiq_xButtonSetCurrentAsJogTarget := FALSE;

		(* generate additional output for the frame FR_CurrentModule *)
		vpq_sCurrentModuleReaction := TPL.FC_ReactionToString(iq_stReaction := vpq_stCurrentModuleStandardInterface.i_stReaction);

		CurrentModuleCmdTable();
	END_IF(* xPointerExceptionActive *)
(****************************************************************************************************************************************************)
END_CASE

IF(NOT xPointerExceptionActive) THEN
	(* point to call additional visualization controllers *)

	(* from Vis_ActiveExceptionList to Vis_ExceptionDetails *)
	IF(vpiq_udiExceptionListGoToDetailsOfLine <> 0) THEN
		IF(vpiq_udiExceptionListGoToDetailsOfLine > 0 AND vpiq_udiExceptionListGoToDetailsOfLine <= 10) THEN
			udiExceptionListDetailsSelectIndex := vpiq_udiExceptionListIndexMin + vpiq_udiExceptionListGoToDetailsOfLine - 1;
		END_IF
		vpiq_udiExceptionListGoToDetailsOfLine := 0;
	END_IF
	
	(* exception handling *)
	vpiq_fbVisContExHandling(	i_xEnable							:= vpq_xDoEnable,
								i_pstMachineStandardItf				:= ADR(SR_MainMachine.stMachineInterface),
								i_pstCurrentStandardItf				:= pstCurrent,
								i_xUpdateData						:= xUpdateForOtherFBs,
								i_udiNumberOfExceptions				:= vpq_udiNumberOfExceptions,
								iq_stExceptionList					:= G_stExceptionList,
								iq_stLogDataList					:= G_stLogDataList,
								iq_astExceptionListCopy				:= astExceptionListCopy,
								iq_udiExceptionDetailsSelectIndex	:= udiExceptionListDetailsSelectIndex,
								q_udiSetAsCurrentModule				=> udiSetAsCurrentModule);
						
	SetCurrentModule();

	(* module specific vis controllers are called inside this action *)
	ModuleVisController();


	(* End of area for vis control fbs of different module types *)
	xUpdateForOtherFBs := FALSE;
END_IF

(* Detect change of OpMode for AxisModule *)
DetectOpModeChange();

ACTION CallTestErrors:
TPL.FC_SetException(i_xExceptionActive := vpiq_xTestUserException1,
					iq_stException := stUserException1,
					iq_stExceptionList := G_stExceptionList,
					iq_stLogDataList := G_stLogDataList);
IF vpiq_xTestUserException1 AND NOT xTestUserException1Old AND (fbLoggerPoint.etLogLevel >= APL.ET_LogLevel.Exception) THEN
	fbLoggerPoint.AddLogEntry(	i_etLogLevel	:= APL.ET_LogLevel.Exception,
								i_etDiag		:= stUserException1.etDiag,
								i_udiDiagExt	:= stUserException1.udiDiagExt,
								i_sMessage		:= stUserException1.sMsg,
								q_etDiag		=> ,
								q_etDiagExt		=> );
END_IF
xTestUserException1Old := vpiq_xTestUserException1; 
	
TPL.FC_SetException(i_xExceptionActive := vpiq_xTestUserException2,
					iq_stException := stUserException2,
					iq_stExceptionList := G_stExceptionList,
					iq_stLogDataList := G_stLogDataList);
IF vpiq_xTestUserException2 AND NOT xTestUserException2Old AND (fbLoggerPoint.etLogLevel >= APL.ET_LogLevel.Exception) THEN
	fbLoggerPoint.AddLogEntry(	i_etLogLevel	:= APL.ET_LogLevel.Exception,
								i_etDiag		:= stUserException2.etDiag,
								i_udiDiagExt	:= stUserException2.udiDiagExt,
								i_sMessage		:= stUserException2.sMsg,
								q_etDiag		=> ,
								q_etDiagExt		=> );
END_IF
xTestUserException2Old := vpiq_xTestUserException2;
	
TPL.FC_SetException(i_xExceptionActive := vpiq_xTestUserException3,
					iq_stException := stUserException3,
					iq_stExceptionList := G_stExceptionList,
					iq_stLogDataList := G_stLogDataList);
IF vpiq_xTestUserException3 AND NOT xTestUserException3Old AND (fbLoggerPoint.etLogLevel >= APL.ET_LogLevel.Exception) THEN
	fbLoggerPoint.AddLogEntry(	i_etLogLevel	:= APL.ET_LogLevel.Exception,
								i_etDiag		:= stUserException3.etDiag,
								i_udiDiagExt	:= stUserException3.udiDiagExt,
								i_sMessage		:= stUserException3.sMsg,
								q_etDiag		=> ,
								q_etDiagExt		=> );
END_IF
xTestUserException3Old := vpiq_xTestUserException3;
	
TPL.FC_SetException(i_xExceptionActive := (vpiq_xTestUserException4 OR vpiq_fbAxisModuleVisController.q_xSimulateExceptionStopEndOfCycle),
					iq_stException := stUserException4,
					iq_stExceptionList := G_stExceptionList,
					iq_stLogDataList := G_stLogDataList);
IF (vpiq_xTestUserException4 OR vpiq_fbAxisModuleVisController.q_xSimulateExceptionStopEndOfCycle) AND NOT xTestUserException4Old AND (fbLoggerPoint.etLogLevel >= APL.ET_LogLevel.Exception) THEN
	fbLoggerPoint.AddLogEntry(	i_etLogLevel	:= APL.ET_LogLevel.Exception,
								i_etDiag		:= stUserException4.etDiag,
								i_udiDiagExt	:= stUserException4.udiDiagExt,
								i_sMessage		:= stUserException4.sMsg,
								q_etDiag		=> ,
								q_etDiagExt		=> );
END_IF
xTestUserException4Old := (vpiq_xTestUserException4 OR vpiq_fbAxisModuleVisController.q_xSimulateExceptionStopEndOfCycle);
	
TPL.FC_SetException(i_xExceptionActive := vpiq_xTestUserException5,
					iq_stException := stUserException5,
					iq_stExceptionList := G_stExceptionList,
					iq_stLogDataList := G_stLogDataList);
IF vpiq_xTestUserException5 AND NOT xTestUserException5Old AND (fbLoggerPoint.etLogLevel >= APL.ET_LogLevel.Exception) THEN
	fbLoggerPoint.AddLogEntry(	i_etLogLevel	:= APL.ET_LogLevel.Exception,
								i_etDiag		:= stUserException5.etDiag,
								i_udiDiagExt	:= stUserException5.udiDiagExt,
								i_sMessage		:= stUserException5.sMsg,
								q_etDiag		=> ,
								q_etDiagExt		=> );
END_IF
xTestUserException5Old := vpiq_xTestUserException5;
END_ACTION

ACTION CrankModuleVis:
IF NOT SR_CharlyModule.stCrankModuleItf.stCrank.xCrankLeft THEN
	vpq_xFrameSetCrankLeftInvisible := TRUE; 
ELSE
	vpq_xFrameSetCrankLeftInvisible := FALSE;
END_IF
END_ACTION

ACTION CurrentModuleCmdTable:
(* Find the active CMD table *)
vpq_udiNumberOfCmdStepsModule :=  0; (* Default values, for security *)
pstEQCMDTableListEntry := 0;
pstEQCMDTable := 0;
IF (vpq_stCurrentModuleStandardInterface.q_diCMDActive <> 0 AND 
	vpq_stCurrentModuleStandardInterface.iq_stExt.udiNumberOfCMDTables > 0 AND 
	vpq_stCurrentModuleStandardInterface.iq_stExt.pstListofCMDTables <> 0) THEN
	
	FOR udiTmp2 := 1 TO vpq_stCurrentModuleStandardInterface.iq_stExt.udiNumberOfCMDTables DO
		pstEQCMDTableListEntry := vpq_stCurrentModuleStandardInterface.iq_stExt.pstListofCMDTables +  UDINT_TO_DWORD((udiTmp2-1)*SIZEOF(pstEQCMDTableListEntry^));
		IF(pstEQCMDTableListEntry^.diCMD = vpq_stCurrentModuleStandardInterface.q_diCMDActive) THEN (* Found *)
			vpq_udiNumberOfCmdStepsModule := pstEQCMDTableListEntry^.udiNumberOfCmdSteps;
			pstEQCMDTable := pstEQCMDTableListEntry^.pstCMDTable;
			vpq_sCmdTitleModule := pstEQCMDTableListEntry^.sTitle;
			EXIT;
		END_IF
	END_FOR
END_IF

(*Command steps > 10 and index changed??*)
IF vpq_udiNumberOfCmdStepsModule <> udiEQTableIndexOld OR udiEQTableStepCountOld <> vpq_udiNumberOfCmdStepsModule THEN
														(*More than 10 steps ??*)
	IF (vpiq_udiIndexMinModule + 9 < vpq_udiNumberOfCmdStepsModule) THEN
		udiEQTableIndexMax := vpiq_udiIndexMinModule + 9;
	ELSE
		udiEQTableIndexMax := vpq_udiNumberOfCmdStepsModule;
	END_IF
														(*Additional safety check*)
	IF (vpiq_udiIndexMinModule < 1) OR (vpiq_udiIndexMinModule > vpq_udiNumberOfCmdStepsModule) THEN
		vpiq_udiIndexMinModule :=1;
		udiEQTableIndexMax := 10;
	END_IF

	udiEQTableIndexOld := vpiq_udiIndexMinModule;
	udiEQTableStepCountOld := vpq_udiNumberOfCmdStepsModule;
END_IF (*vpiq_udiIndexMinModule <> udiEQTableIndexOld*)

vpq_xDisableScrollUpModule := NOT (vpiq_udiIndexMinModule > 1);
vpq_xDisableScrollDownModule := NOT (vpiq_udiIndexMinModule + 9 < vpq_udiNumberOfCmdStepsModule);

IF(pstEQCMDTable <> 0) THEN
	FOR udiCounter := udiEQTableIndexOld TO udiEQTableIndexMax DO
		pstEQCMDTableEntry := pstEQCMDTable +  UDINT_TO_DWORD(((udiCounter-1) * SIZEOF(pstEQCMDTable^)));
		vpq_astActualCmdTableModule[udiCounter - udiEQTableIndexOld + 1] := pstEQCMDTableEntry^;
	END_FOR
	FOR udiCounter := udiEQTableIndexMax + 1 TO udiEQTableIndexOld + 9 DO
		vpq_astActualCmdTableModule[udiCounter - udiEQTableIndexOld + 1] := c_stEmptyCmdTableStep;
	END_FOR
	vpq_xDisplayCmdTable := TRUE;
ELSE
	vpq_xDisplayCmdTable := FALSE;
END_IF
END_ACTION

ACTION DetectOpModeChange:
IF (vpiq_fbAxisModuleVisController.i_pstCurrentStandardItf <> 0) THEN
	IF (v_diLastOpMode <> vpiq_fbAxisModuleVisController.i_pstCurrentStandardItf^.q_diCmdActive) THEN
		v_diLastOpMode := vpiq_fbAxisModuleVisController.i_pstCurrentStandardItf^.q_diCmdActive;
		CASE (v_diLastOpMode) OF
			AXM.ET_Cmd.Homing:
				v_xHomeModeActive := TRUE;
				v_xManualModeActive := FALSE;
				v_xMultiCamCSActive := FALSE;
				v_xMultiCamWSActive := FALSE;
				v_xEndlessActive := FALSE;
				v_xEndlessILSActive := FALSE;
				v_xPositioningActive := FALSE;
				v_xBrakeActive := FALSE;
				v_xAdditionalCSActive := FALSE;
				v_xAdditionalWSActive := FALSE;		
			AXM.ET_Cmd.Manual:
				v_xHomeModeActive := FALSE;
				v_xManualModeActive := TRUE;
				v_xMultiCamCSActive := FALSE;
				v_xMultiCamWSActive := FALSE;
				v_xEndlessActive := FALSE;
				v_xEndlessILSActive := FALSE;
				v_xPositioningActive := FALSE;
				v_xBrakeActive := FALSE;
				v_xAdditionalCSActive := FALSE;
				v_xAdditionalWSActive := FALSE;
			
			AXM.ET_Cmd.CamCs:
				v_xHomeModeActive := FALSE;
				v_xManualModeActive := FALSE;
				v_xMultiCamCSActive := TRUE;
				v_xMultiCamWSActive := FALSE;
				v_xEndlessActive := FALSE;
				v_xEndlessILSActive := FALSE;
				v_xPositioningActive := FALSE;
				v_xBrakeActive := FALSE;
				v_xAdditionalCSActive := FALSE;
				v_xAdditionalWSActive := FALSE;
			
			AXM.ET_Cmd.CamWs:
				v_xHomeModeActive := FALSE;
				v_xManualModeActive := FALSE;
				v_xMultiCamCSActive := FALSE;
				v_xMultiCamWSActive := TRUE;
				v_xEndlessActive := FALSE;
				v_xEndlessILSActive := FALSE;
				v_xPositioningActive := FALSE;
				v_xBrakeActive := FALSE;
				v_xAdditionalCSActive := FALSE;
				v_xAdditionalWSActive := FALSE;
			
			AXM.ET_Cmd.Endless:
				v_xHomeModeActive := FALSE;
				v_xManualModeActive := FALSE;
				v_xMultiCamCSActive := FALSE;
				v_xMultiCamWSActive := FALSE;
				v_xEndlessActive := TRUE;
				v_xEndlessILSActive := FALSE;
				v_xPositioningActive := FALSE;
				v_xBrakeActive := FALSE;
				v_xAdditionalCSActive := FALSE;
				v_xAdditionalWSActive := FALSE;
			
			AXM.ET_Cmd.EndlessIls:
				v_xHomeModeActive := FALSE;
				v_xManualModeActive := FALSE;
				v_xMultiCamCSActive := FALSE;
				v_xMultiCamWSActive := FALSE;
				v_xEndlessActive := FALSE;
				v_xEndlessILSActive := TRUE;
				v_xPositioningActive := FALSE;
				v_xBrakeActive := FALSE;
				v_xAdditionalCSActive := FALSE;
				v_xAdditionalWSActive := FALSE;
			
			AXM.ET_Cmd.Positioning:
				v_xHomeModeActive := FALSE;
				v_xManualModeActive := FALSE;
				v_xMultiCamCSActive := FALSE;
				v_xMultiCamWSActive := FALSE;
				v_xEndlessActive := FALSE;
				v_xEndlessILSActive := FALSE;
				v_xPositioningActive := TRUE;
				v_xBrakeActive := FALSE;
				v_xAdditionalCSActive := FALSE;
				v_xAdditionalWSActive := FALSE;
			
			AXM.ET_Cmd.BrakeRelease:
				v_xHomeModeActive := FALSE;
				v_xManualModeActive := FALSE;
				v_xMultiCamCSActive := FALSE;
				v_xMultiCamWSActive := FALSE;
				v_xEndlessActive := FALSE;
				v_xEndlessILSActive := FALSE;
				v_xPositioningActive := FALSE;
				v_xBrakeActive := TRUE;
				v_xAdditionalCSActive := FALSE;
				v_xAdditionalWSActive := FALSE;
			
			AXM.ET_Cmd.AdditionalCs:
				v_xHomeModeActive := FALSE;
				v_xManualModeActive := FALSE;
				v_xMultiCamCSActive := FALSE;
				v_xMultiCamWSActive := FALSE;
				v_xEndlessActive := FALSE;
				v_xEndlessILSActive := FALSE;
				v_xPositioningActive := FALSE;
				v_xBrakeActive := FALSE;
				v_xAdditionalCSActive := TRUE;
				v_xAdditionalWSActive := FALSE;
			
			AXM.ET_Cmd.AdditionalWs:
				v_xHomeModeActive := FALSE;
				v_xManualModeActive := FALSE;
				v_xMultiCamCSActive := FALSE;
				v_xMultiCamWSActive := FALSE;
				v_xEndlessActive := FALSE;
				v_xEndlessILSActive := FALSE;
				v_xPositioningActive := FALSE;
				v_xBrakeActive := FALSE;
				v_xAdditionalCSActive := FALSE;
				v_xAdditionalWSActive := TRUE;
		END_CASE
	END_IF
END_IF
END_ACTION

ACTION ExceptionVis:
stActiveReactions := vpq_stMachineInterface.i_stReaction;

fbCopyExceptionList(i_xEnable					:= TRUE,
					i_xCopy						:= TRUE,
					i_timElapsedTimeUpdate		:= T#1S, (* update todElapsedTime every seccond, is fast enough for user interface *)
					iq_stExceptionList			:= G_stExceptionList,
					iq_astException				:= astExceptionListCopy,
					iq_udiNumberOfExceptions	:= vpq_udiNumberOfExceptions,
					q_xActive					=> ,
					q_xReady					=> ,
					q_etDiag					=> ,
					q_etDiagExt					=> );

IF vpiq_xReactionUp THEN
	vpq_udiReactionIndexMin := vpq_udiReactionIndexMin + 1;
	vpiq_xReactionUp:=FALSE;
ELSIF vpiq_xReactionDown THEN
	vpq_udiReactionIndexMin := vpq_udiReactionIndexMin - 1;
	vpiq_xReactionDown:=FALSE;
END_IF

IF vpq_udiReactionIndexMin <> udiReactionIndexOld THEN
														(*More than 10 steps ??*)
	IF (vpq_udiReactionIndexMin + 9 < TPL.Gc_udiMaxNumberOfReactions) THEN
		udiReactionIndexMax := vpq_udiReactionIndexMin + 9;
	ELSE
		udiReactionIndexMax := TPL.Gc_udiMaxNumberOfReactions;
	END_IF
														(*Additional safety check*)
	IF (vpq_udiReactionIndexMin < 1) THEN
		vpq_udiReactionIndexMin := 1;
		udiReactionIndexMax := 10;
	ELSIF (vpq_udiReactionIndexMin > TPL.Gc_udiMaxNumberOfReactions - 9) THEN
		vpq_udiReactionIndexMin := TPL.Gc_udiMaxNumberOfReactions - 9;
		udiReactionIndexMax := 10;
	END_IF

	udiReactionIndexOld := vpq_udiReactionIndexMin;
END_IF

IF TPL.Gc_udiMaxNumberOfReactions < 10 THEN
	udiMaxValue := TPL.Gc_udiMaxNumberOfReactions;
ELSE
	udiMaxValue := 10;
END_IF

FOR udiCount := 1 TO udiMaxValue  DO
	vpq_axReaction[udiCount] := stActiveReactions.axReaction[vpq_udiReactionIndexMin + udiCount - 1];
END_FOR

(*For Displaying the ErrorList-Visualization Vis_ActiveErrorList*)
IF vpiq_udiExceptionListIndexMin < 1 THEN
	vpiq_udiExceptionListIndexMin := 1;
END_IF

IF vpiq_udiExceptionListIndexMin > TPL.Gc_udiMaxNumberOfExceptions - 9 THEN
	vpiq_udiExceptionListIndexMin := TPL.Gc_udiMaxNumberOfExceptions - 9;
END_IF


FOR udiIndex := 1 TO 10 DO
	vpq_astExceptionListTable[udiIndex] := astExceptionListCopy[vpiq_udiExceptionListIndexMin + udiIndex - 1];
	vpq_asReaction [udiIndex] := TPL.FC_ReactionToString(astExceptionListCopy[vpiq_udiExceptionListIndexMin + udiIndex - 1].stReaction);
END_FOR

vpq_udiExceptionListIndexMax := vpiq_udiExceptionListIndexMin + 9;

IF vpq_udiExceptionListIndexMax > vpq_udiNumberOfExceptions - 1  THEN
	vpq_xDisplayScrollDown := TRUE;
ELSE
	vpq_xDisplayScrollDown := FALSE;
END_IF


vpq_sAllActiveReactions:= TPL.FC_ReactionToString(stActiveReactions);
CallTestErrors();

FOR udiCount := 1 TO TPL.Gc_udiMaxNumberOfReactions DO
	IF stActiveReactions.axReaction[udiCount] THEN
		xRedColor	:= TRUE;
		EXIT;
	ELSE
		xRedColor	:= FALSE;
	END_IF
END_FOR

IF xRedColor THEN
	vpq_dwDiagQuitColor := 16#FF0000;
ELSE
	vpq_dwDiagQuitColor := 16#FFFF00;
END_IF

IF vpiq_xButtonShowExtendedTimes AND NOT vpq_xShowExtendedTimes THEN
	vpq_xShowExtendedTimes		:= TRUE;
	vpq_xShowExtended2			:= FALSE;
	vpiq_xButtonShowExtendedTimes := FALSE;
	vpiq_xButtonShowExtended2		:= FALSE;
ELSIF vpiq_xButtonShowExtendedTimes  AND vpq_xShowExtendedTimes THEN
	vpq_xShowExtendedTimes		:= FALSE;
	vpq_xShowExtended2			:= FALSE;
	vpiq_xButtonShowExtendedTimes := FALSE;
	vpiq_xButtonShowExtended2		:= FALSE;
END_IF

IF vpiq_xButtonShowExtended2 AND NOT vpq_xShowExtended2 THEN
	vpq_xShowExtendedTimes		:= FALSE;
	vpq_xShowExtended2			:= TRUE;
	vpiq_xButtonShowExtendedTimes := FALSE;
	vpiq_xButtonShowExtended2		:= FALSE;
ELSIF vpiq_xButtonShowExtended2 AND vpq_xShowExtended2 THEN
	vpq_xShowExtendedTimes		:= FALSE;
	vpq_xShowExtended2			:= FALSE;
	vpiq_xButtonShowExtendedTimes := FALSE;
	vpiq_xButtonShowExtended2		:= FALSE;
END_IF
END_ACTION

ACTION InitTestExceptions:
stUserException1.etDiag														:= GD.ET_Diag.ExecutionAborted;
stUserException1.udiDiagExt													:= ET_DiagExt.Exception1FromVis;
stUserException1.sDiagExt													:= FC_EtDiagExtToString(ET_DiagExt.Exception1FromVis);
stUserException1.sMsg														:= 'Test Exception 1 from visualization - TPL.ET_Reaction.AsyncStop';
stUserException1.udiModuleId												:= vpq_stMachineInterface.i_udiModuleId;
stUserException1.sModuleName												:= vpq_stMachineInterface.i_sModuleName;
stUserException1.etSource													:= TPL.ET_ExceptionSource.Vis;
stUserException1.timDelayTime												:= T#0MS;
stUserException1.wHmiAttributes												:= 0;
stUserException1.xAutoQuit													:= FALSE;
stUserException1.stReaction.axReaction[TPL.ET_Reaction.AsyncStop]			:= TRUE;

stUserException2.etDiag														:= GD.ET_Diag.ExecutionAborted;
stUserException2.udiDiagExt													:= ET_DiagExt.Exception2FromVis;
stUserException2.sDiagExt													:= FC_EtDiagExtToString(ET_DiagExt.Exception2FromVis);
stUserException2.sMsg														:= 'Test Exception 2 from visualization - TPL.ET_Reaction.SyncStopEL';
stUserException2.udiModuleId												:= vpq_stMachineInterface.i_udiModuleId;
stUserException2.sModuleName												:= vpq_stMachineInterface.i_sModuleName;
stUserException2.etSource													:= TPL.ET_ExceptionSource.Vis;
stUserException2.timDelayTime												:= T#0MS;
stUserException2.wHmiAttributes												:= 0;
stUserException2.xAutoQuit													:= FALSE;
stUserException2.stReaction.axReaction[TPL.ET_Reaction.SyncStopEL]			:= TRUE;

stUserException3.etDiag														:= GD.ET_Diag.ExecutionAborted;
stUserException3.udiDiagExt													:= ET_DiagExt.Exception3FromVis;
stUserException3.sDiagExt													:= FC_EtDiagExtToString(ET_DiagExt.Exception3FromVis);
stUserException3.sMsg														:= 'Test Exception 3 from visualization - TPL.ET_Reaction.SyncStopEH';
stUserException3.udiModuleId												:= vpq_stMachineInterface.i_udiModuleId;
stUserException3.sModuleName												:= vpq_stMachineInterface.i_sModuleName;
stUserException3.etSource													:= TPL.ET_ExceptionSource.Vis;
stUserException3.timDelayTime												:= T#0MS;
stUserException3.wHmiAttributes												:= 0;
stUserException3.xAutoQuit													:= FALSE;
stUserException3.stReaction.axReaction[TPL.ET_Reaction.SyncStopEH]			:= TRUE;

stUserException4.etDiag														:= GD.ET_Diag.ExecutionAborted;
stUserException4.udiDiagExt													:= ET_DiagExt.Exception4FromVis;
stUserException4.sDiagExt													:= FC_EtDiagExtToString(ET_DiagExt.Exception4FromVis);
stUserException4.sMsg														:= 'Test Exception 4 from visualization - TPL.ET_Reaction.StopEndOfCycle';
stUserException4.udiModuleId												:= vpq_stMachineInterface.i_udiModuleId;
stUserException4.sModuleName												:= vpq_stMachineInterface.i_sModuleName;
stUserException4.etSource													:= TPL.ET_ExceptionSource.Vis;
stUserException4.timDelayTime												:= T#0MS;
stUserException4.wHmiAttributes												:= 0;
stUserException4.xAutoQuit													:= FALSE;
stUserException4.stReaction.axReaction[TPL.ET_Reaction.StopEndOfCycle]		:= TRUE;

stUserException5.etDiag														:= GD.ET_Diag.ExecutionAborted;
stUserException5.udiDiagExt													:= ET_DiagExt.Exception5FromVis;
stUserException5.sDiagExt													:= FC_EtDiagExtToString(ET_DiagExt.Exception5FromVis);
stUserException5.sMsg														:= 'Test Exception 5 from visualization - TPL.ET_Reaction.MainsContactorOff';
stUserException5.udiModuleId												:= vpq_stMachineInterface.i_udiModuleId;
stUserException5.sModuleName												:= vpq_stMachineInterface.i_sModuleName;
stUserException5.etSource													:= TPL.ET_ExceptionSource.Vis;
stUserException5.timDelayTime												:= T#0MS;
stUserException5.wHmiAttributes												:= 0;
stUserException5.xAutoQuit													:= FALSE;
stUserException5.stReaction.axReaction[TPL.ET_Reaction.MainsContactorOff]	:= TRUE;
stUserException5.stReaction.axReaction[TPL.ET_Reaction.StopEndOfCycle]		:= TRUE;
END_ACTION

ACTION LoggerVis:
(*For Displaying the LoggerList-Visualization Vis_Logger*)
IF vpiq_udiLogDataListIndexMin < 1 THEN
	vpiq_udiLogDataListIndexMin := 1;
END_IF

IF vpiq_udiLogDataListIndexMin > TPL.Gc_udiMaxNumberOfLogData - 11 THEN
	vpiq_udiLogDataListIndexMin := TPL.Gc_udiMaxNumberOfLogData - 11;
END_IF

FOR udiIndex2 := 1 TO 12 DO
	vpq_astLogDataTableAscii[udiIndex2] := G_stLogDataListAscii.astLogData[vpiq_udiLogDataListIndexMin + udiIndex2 - 1];

	IF G_stLogDataListAscii.astLogData[vpiq_udiLogDataListIndexMin + udiIndex2 - 1].asAsciiData[1]= 'Cmd come' THEN
			vpq_astLogDataTable[udiIndex2].etReason:= TPL. ET_LogDataFilter.CmdCome;
	ELSIF G_stLogDataListAscii.astLogData[vpiq_udiLogDataListIndexMin + udiIndex2 - 1].asAsciiData[1]= 'Cmd go' THEN
			vpq_astLogDataTable[udiIndex2].etReason:= TPL.ET_LogDataFilter.CmdGo;
	ELSIF G_stLogDataListAscii.astLogData[vpiq_udiLogDataListIndexMin + udiIndex2 - 1].asAsciiData[1]= 'StartStep come' THEN
			vpq_astLogDataTable[udiIndex2].etReason:= TPL.ET_LogDataFilter.StartStepCome;
	ELSIF G_stLogDataListAscii.astLogData[vpiq_udiLogDataListIndexMin + udiIndex2 - 1].asAsciiData[1]= 'StartStep go' THEN
			vpq_astLogDataTable[udiIndex2].etReason:= TPL.ET_LogDataFilter.StartStepGo;
	ELSIF G_stLogDataListAscii.astLogData[vpiq_udiLogDataListIndexMin + udiIndex2 - 1].asAsciiData[1]= 'Reaction come' THEN
			vpq_astLogDataTable[udiIndex2].etReason:= TPL.ET_LogDataFilter.ReactionCome;
	ELSIF G_stLogDataListAscii.astLogData[vpiq_udiLogDataListIndexMin + udiIndex2 - 1].asAsciiData[1]= 'Reaction go' THEN
			vpq_astLogDataTable[udiIndex2].etReason:= TPL.ET_LogDataFilter.ReactionGo;
	ELSIF G_stLogDataListAscii.astLogData[vpiq_udiLogDataListIndexMin + udiIndex2 - 1].asAsciiData[1]= 'Exception quit' THEN
			vpq_astLogDataTable[udiIndex2].etReason:= TPL.ET_LogDataFilter.ExceptionQuit;
	ELSIF G_stLogDataListAscii.astLogData[vpiq_udiLogDataListIndexMin + udiIndex2 - 1].asAsciiData[1]= 'Exception come' THEN
			vpq_astLogDataTable[udiIndex2].etReason := TPL.ET_LogDataFilter.ExceptionCome;
	ELSIF G_stLogDataListAscii.astLogData[vpiq_udiLogDataListIndexMin + udiIndex2 - 1].asAsciiData[1]= 'Exception autoquit' THEN
			vpq_astLogDataTable[udiIndex2].etReason:= TPL.ET_LogDataFilter.ExceptionAutoQuit;
	ELSIF G_stLogDataListAscii.astLogData[vpiq_udiLogDataListIndexMin + udiIndex2 - 1].asAsciiData[1]= 'User entry' THEN
			vpq_astLogDataTable[udiIndex2].etReason:= TPL.ET_LogDataFilter.User;
	ELSE
		vpq_astLogDataTable[udiIndex2].etReason:= TPL.ET_LogDataFilter.None;
	END_IF
	vpq_astLogDataTable[udiIndex2].dateDate 		:= STRING_TO_DATE(G_stLogDataListAscii.astLogData[vpiq_udiLogDataListIndexMin + udiIndex2 - 1].asAsciiData[2]);
	vpq_astLogDataTable[udiIndex2].todTime			:= STRING_TO_TOD(G_stLogDataListAscii.astLogData[vpiq_udiLogDataListIndexMin + udiIndex2 - 1].asAsciiData[3]);
	vpq_astLogDataTable[udiIndex2].udiModuleId		:= STRING_TO_UDINT(G_stLogDataListAscii.astLogData[vpiq_udiLogDataListIndexMin + udiIndex2 - 1].asAsciiData[4]);
	vpq_astLogDataTable[udiIndex2].sModuleName		:= G_stLogDataListAscii.astLogData[vpiq_udiLogDataListIndexMin + udiIndex2 - 1].asAsciiData[5];
	vpq_astLogDataTable[udiIndex2].diCMD			:= STRING_TO_DINT(G_stLogDataListAscii.astLogData[vpiq_udiLogDataListIndexMin + udiIndex2 - 1].asAsciiData[6]);
	vpq_astLogDataTable[udiIndex2].diStartStep		:= STRING_TO_DINT(G_stLogDataListAscii.astLogData[vpiq_udiLogDataListIndexMin + udiIndex2 - 1].asAsciiData[7]);

	vpq_astLogDataTable[udiIndex2].etDiag			:= STRING_TO_UDINT(G_stLogDataListAscii.astLogData[vpiq_udiLogDataListIndexMin + udiIndex2 - 1].asAsciiData[8]);
	vpq_astLogDataTable[udiIndex2].udiDiagExt		:= STRING_TO_UDINT(G_stLogDataListAscii.astLogData[vpiq_udiLogDataListIndexMin + udiIndex2 - 1].asAsciiData[10]);
	vpq_astLogDataTable[udiIndex2].sDiagExt			:= G_stLogDataListAscii.astLogData[vpiq_udiLogDataListIndexMin + udiIndex2 - 1].asAsciiData[11];
	vpq_astLogDataTable[udiIndex2].sMsg				:= G_stLogDataListAscii.astLogData[vpiq_udiLogDataListIndexMin + udiIndex2 - 1].asAsciiData[12];
	
	FOR udiIndex3 := 1 TO TPL.Gc_udiMaxNumberOfReactions DO
		IF FIND(G_stLogDataListAscii.astLogData[vpiq_udiLogDataListIndexMin + udiIndex2 - 1].asAsciiData[13], UDINT_TO_STRING(udiIndex3))<>0 THEN
			vpq_astLogDataTable[udiIndex2].stReaction.axReaction[udiIndex3] := TRUE;
		ELSE
			vpq_astLogDataTable[udiIndex2].stReaction.axReaction[udiIndex3] := FALSE;
		END_IF
	END_FOR

	IF    G_stLogDataListAscii.astLogData[vpiq_udiLogDataListIndexMin + udiIndex2 - 1].asAsciiData[14]= '1' THEN
		vpq_astLogDataTable[udiIndex2].etSource:= TPL.ET_ExceptionSource.ModuleController;
	ELSIF G_stLogDataListAscii.astLogData[vpiq_udiLogDataListIndexMin + udiIndex2 - 1].asAsciiData[14]= '2' THEN
		vpq_astLogDataTable[udiIndex2].etSource:= TPL.ET_ExceptionSource.ExceptionHandler;
	ELSIF G_stLogDataListAscii.astLogData[vpiq_udiLogDataListIndexMin + udiIndex2 - 1].asAsciiData[14]= '3' THEN
		vpq_astLogDataTable[udiIndex2].etSource:= TPL.ET_ExceptionSource.Logger;
	ELSIF G_stLogDataListAscii.astLogData[vpiq_udiLogDataListIndexMin + udiIndex2 - 1].asAsciiData[14]= '4' THEN
		vpq_astLogDataTable[udiIndex2].etSource:= TPL.ET_ExceptionSource.Main;
	ELSIF G_stLogDataListAscii.astLogData[vpiq_udiLogDataListIndexMin + udiIndex2 - 1].asAsciiData[14]= '5' THEN
		vpq_astLogDataTable[udiIndex2].etSource:= TPL.ET_ExceptionSource.Vis;
	ELSIF G_stLogDataListAscii.astLogData[vpiq_udiLogDataListIndexMin + udiIndex2 - 1].asAsciiData[14]= '6' THEN
		vpq_astLogDataTable[udiIndex2].etSource:= TPL.ET_ExceptionSource.User;
	ELSIF G_stLogDataListAscii.astLogData[vpiq_udiLogDataListIndexMin + udiIndex2 - 1].asAsciiData[14]= '7' THEN
		vpq_astLogDataTable[udiIndex2].etSource:= TPL.ET_ExceptionSource.NodeModule;
	ELSIF G_stLogDataListAscii.astLogData[vpiq_udiLogDataListIndexMin + udiIndex2 - 1].asAsciiData[14]= '8' THEN
		vpq_astLogDataTable[udiIndex2].etSource:= TPL.ET_ExceptionSource.AxisModule;
	ELSIF G_stLogDataListAscii.astLogData[vpiq_udiLogDataListIndexMin + udiIndex2 - 1].asAsciiData[14]= '9' THEN
		vpq_astLogDataTable[udiIndex2].etSource:= TPL.ET_ExceptionSource.MultiBeltModule;
	ELSIF G_stLogDataListAscii.astLogData[vpiq_udiLogDataListIndexMin + udiIndex2 - 1].asAsciiData[14]= '10' THEN
		vpq_astLogDataTable[udiIndex2].etSource:= TPL.ET_ExceptionSource.SmartInfeedModule;
	ELSIF G_stLogDataListAscii.astLogData[vpiq_udiLogDataListIndexMin + udiIndex2 - 1].asAsciiData[14]= '11' THEN
		vpq_astLogDataTable[udiIndex2].etSource:= TPL.ET_ExceptionSource.RoboticModule;
	ELSIF G_stLogDataListAscii.astLogData[vpiq_udiLogDataListIndexMin + udiIndex2 - 1].asAsciiData[14]= '12' THEN
		vpq_astLogDataTable[udiIndex2].etSource:= TPL.ET_ExceptionSource.UnwinderModule;
	ELSIF G_stLogDataListAscii.astLogData[vpiq_udiLogDataListIndexMin + udiIndex2 - 1].asAsciiData[14]= '13' THEN
		vpq_astLogDataTable[udiIndex2].etSource:= TPL.ET_ExceptionSource.SealingModule;
	ELSIF G_stLogDataListAscii.astLogData[vpiq_udiLogDataListIndexMin + udiIndex2 - 1].asAsciiData[14]= '14' THEN
		vpq_astLogDataTable[udiIndex2].etSource:= TPL.ET_ExceptionSource.AtvModule;
	ELSIF G_stLogDataListAscii.astLogData[vpiq_udiLogDataListIndexMin + udiIndex2 - 1].asAsciiData[14]= '15' THEN
		vpq_astLogDataTable[udiIndex2].etSource:= TPL.ET_ExceptionSource.IlxModule;
	ELSIF G_stLogDataListAscii.astLogData[vpiq_udiLogDataListIndexMin + udiIndex2 - 1].asAsciiData[14]= '16' THEN
		vpq_astLogDataTable[udiIndex2].etSource:= TPL.ET_ExceptionSource.CrankModule;
	ELSIF G_stLogDataListAscii.astLogData[vpiq_udiLogDataListIndexMin + udiIndex2 - 1].asAsciiData[14]= '17' THEN
		vpq_astLogDataTable[udiIndex2].etSource:= TPL.ET_ExceptionSource.ValveModule;
	ELSIF G_stLogDataListAscii.astLogData[vpiq_udiLogDataListIndexMin + udiIndex2 - 1].asAsciiData[14]= '18' THEN
		vpq_astLogDataTable[udiIndex2].etSource:= TPL.ET_ExceptionSource.CapperModule;
	ELSE
		vpq_astLogDataTable[udiIndex2].etSource:= TPL.ET_ExceptionSource.None;
	END_IF
	
	vpq_astLogDataTable[udiIndex2].xAutoQuit	:= STRING_TO_BOOL(G_stLogDataListAscii.astLogData[vpiq_udiLogDataListIndexMin + udiIndex2 - 1].asAsciiData[15]);
END_FOR


vpq_udiLogDataListIndexMax := vpiq_udiLogDataListIndexMin + 11;

vpiq_udiNumberOfLogData := G_stLogDataListAscii.udiNumberOfLogData;
IF vpq_udiLogDataListIndexMax > G_stLogDataListAscii.udiNumberOfLogData - 1  THEN
	vpq_xLogDataScrollDown := TRUE;

ELSE
	vpq_xLogDataScrollDown := FALSE;
END_IF

IF vpiq_xButtonLogDataListDetails AND NOT vpq_xShowLogDataListDetails THEN
	vpq_xShowLogDataListDetails				:= TRUE;
	vpiq_xButtonLogDataListDetails			:= FALSE;
ELSIF vpiq_xButtonLogDataListDetails AND vpq_xShowLogDataListDetails THEN
	vpq_xShowLogDataListDetails				:= FALSE;
	vpiq_xButtonLogDataListDetails			:= FALSE;
END_IF
END_ACTION

ACTION MainPageCmdTable:
(* Find the current table*)
vpq_udiNumberOfCmdStepsModule		:= 0; (* Default values, for security *)
pstEQCMDTableListEntry	:= 0;
pstEQCMDTable			:= 0;

IF(vpq_stMachineInterface.q_diCmdActive <> 0 AND vpq_stMachineInterface.iq_stExt.udiNumberOfCmdTables > 0 AND vpq_stMachineInterface.iq_stExt.pstListofCMDTables <> 0) THEN
	FOR udiTmp2 := 1 TO vpq_stMachineInterface.iq_stExt.udiNumberOfCMDTables DO
		pstEQCMDTableListEntry := vpq_stMachineInterface.iq_stExt.pstListofCMDTables +  UDINT_TO_DWORD((udiTmp2-1)*SIZEOF(pstEQCMDTableListEntry^));
		IF(pstEQCMDTableListEntry^.diCMD = vpq_stMachineInterface.q_diCmdActive) THEN (* Found *)
			vpq_udiNumberOfCmdStepsModule := pstEQCMDTableListEntry^.udiNumberOfCmdSteps;
			vpq_udiNumberOfCmdStepsMain := vpq_udiNumberOfCmdStepsModule;
			pstEQCMDTable := pstEQCMDTableListEntry^.pstCMDTable;
			vpq_sCmdTitelMain := pstEQCMDTableListEntry^.sTitle;
			EXIT;
		END_IF
	END_FOR
END_IF

(***********************************************************************************************************************)
(* Check the limits of the Vis/ shown table *)
udiIndexOldMainTable := 0;
IF vpiq_udiIndexMinMain <> udiIndexOldMainTable THEN
														(*More than 10 steps ??*)
	IF (vpiq_udiIndexMinMain + 9 < vpq_udiNumberOfCmdStepsMain) THEN
		udiIndexMaxMainTable := vpiq_udiIndexMinMain + 9;
	ELSE
		udiIndexMaxMainTable := vpq_udiNumberOfCmdStepsMain;
	END_IF
														(*Additional safety check*)
	IF (vpiq_udiIndexMinMain < 1) OR (vpiq_udiIndexMinMain > vpq_udiNumberOfCmdStepsMain) THEN
		vpiq_udiIndexMinMain :=1;
		udiIndexMaxMainTable := 10;
	END_IF

	udiIndexOldMainTable := vpiq_udiIndexMinMain;
END_IF (*udiEQMainTableIndexMin <> udiEQMainTableIndexOld*)

vpq_xDisableScrollUpMain	:= NOT (vpiq_udiIndexMinMain > 1);
vpq_xDisableScrollDownMain	:= NOT (vpiq_udiIndexMinMain + 9 < vpq_udiNumberOfCmdStepsMain) ;

(***********************************************************************************************************************)
(*Refresh the values in the table if more then "Max commands" should be shown!*)
IF(pstEQCMDTable <> 0) THEN
	FOR udiCounter := udiIndexOldMainTable TO udiIndexMaxMainTable DO
		pstEQCMDTableEntry := pstEQCMDTable +  UDINT_TO_DWORD(((udiCounter-1) * SIZEOF(pstEQCMDTable^)));
		vpq_astActualCmdTableMain[udiCounter - udiIndexOldMainTable + 1] := pstEQCMDTableEntry^;
	END_FOR
	FOR udiCounter := udiIndexMaxMainTable + 1 TO udiIndexOldMainTable + 9 DO
		vpq_astActualCmdTableMain[udiCounter - udiIndexOldMainTable + 1] := c_stEmptyCmdTableStep;
	END_FOR
END_IF
END_ACTION

ACTION ModuleNavigationIn:
(* Navigation *)

(* 2D navigation *)
IF(vpiq_xNavUp OR vpiq_xNavDown OR vpiq_xNavLeft OR vpiq_xNavRight) THEN
	IF vpiq_xNavRight THEN
		(* Move the the next module on the same level *)
		IF audiHierarchy[udiCurrentLevel] + 1 <= udiCurrentLevelSize + udiCurrentNumberOfControlModules  THEN
			audiHierarchy[udiCurrentLevel] := audiHierarchy[udiCurrentLevel] + 1;
			IF audiHierarchy[udiCurrentLevel]  > udiCurrentLevelSize THEN
				udiControlModuleSelectedInLevel	:= udiCurrentLevel;
				vpq_udiActiveControlModuleNumber:= audiHierarchy[udiCurrentLevel]-udiCurrentLevelSize;
			END_IF
		END_IF
	END_IF
	IF vpiq_xNavLeft THEN
		(* Move the the previous module on the same level *)
		IF audiHierarchy[udiCurrentLevel] -1 >= 1 THEN
			audiHierarchy[udiCurrentLevel] := audiHierarchy[udiCurrentLevel] - 1;
			vpq_udiActiveControlModuleNumber:= audiHierarchy[udiCurrentLevel]-udiCurrentLevelSize;
			IF audiHierarchy[udiCurrentLevel] <= udiCurrentLevelSize THEN
				udiControlModuleSelectedInLevel	:= 0;
				vpq_udiActiveControlModuleNumber:= 0;
			END_IF
		END_IF (* ELSE ignore *)
	END_IF
	IF vpiq_xNavUp THEN
		(* Move one level up *)
		udiControlModuleSelectedInLevel := 0;
		vpq_udiActiveControlModuleNumber:= 0;
		IF udiCurrentLevel - 1 >= 1 THEN
			udiCurrentLevel := udiCurrentLevel - 1;
		END_IF (* ELSE ignore *)
	END_IF
	IF vpiq_xNavDown THEN
		(* Move one level down *)
		IF (udiCurrentLevel + 1 <= c_udiMaxHierarchyLevels) AND (xCurrentHasSubModules OR xCurrentHasControlModules) THEN
			udiCurrentLevel := udiCurrentLevel + 1;
			audiHierarchy[udiCurrentLevel] := 1;
			IF NOT xCurrentHasSubModules AND xCurrentHasControlModules THEN
				udiControlModuleSelectedInLevel := udiCurrentLevel;
				vpq_udiActiveControlModuleNumber:= audiHierarchy[udiCurrentLevel];
			ELSE
				udiControlModuleSelectedInLevel	:= 0;
				vpq_udiActiveControlModuleNumber:= 0;
			END_IF

		END_IF (* ELSE ignore *)
	END_IF

	vpiq_xNavUp		:= FALSE;
	vpiq_xNavDown	:= FALSE;
	vpiq_xNavLeft	:= FALSE;
	vpiq_xNavRight	:= FALSE;
	
	xUpdateData := TRUE;
END_IF (* End 2D navbutton hit *)

(* Direct navigation (on level 2 and 3) *)
(* Module level *)
IF vpiq_axModuleList[1] OR vpiq_axModuleList[2] OR vpiq_axModuleList[3] OR vpiq_axModuleList[4] OR vpiq_axModuleList[5] OR
   vpiq_axControlModuleList[1] OR vpiq_axControlModuleList[2] OR vpiq_axControlModuleList[3] OR vpiq_axControlModuleList[4] OR vpiq_axControlModuleList[5] THEN
	udiCurrentLevel := 2;
	udiCurrentLevel := 2;
	FOR udiTmp := 1 TO 5 DO
		(*select an equipment module via the buttons on level 2*)
		IF(vpiq_axModuleList[udiTmp]) THEN
			audiHierarchy[udiCurrentLevel] := udiTmp + udiMinModuleList - 1;
			vpiq_axModuleList[udiTmp] := FALSE;
			udiControlModuleSelectedInLevel := 0;
			vpq_udiActiveControlModuleNumber:= 0;
		END_IF
		(*select a control module via the buttons on level 2*)
		IF vpiq_axControlModuleList[udiTmp] THEN
			audiHierarchy[udiCurrentLevel] := udiTmp + udiMinModuleList - 1;
			udiControlModuleSelectedInLevel	:= udiCurrentLevel;
			vpiq_axControlModuleList[udiTmp] := FALSE;
		END_IF
	END_FOR
	xUpdateData := TRUE;
END_IF
IF vpiq_xModuleListDown THEN
	vpiq_xModuleListDown := FALSE;
	IF(udiMinModuleList > 1) THEN
		udiMinModuleList := udiMinModuleList - 1;
	END_IF
	xUpdateData := TRUE;
END_IF
IF vpiq_xModuleListUp THEN
	vpiq_xModuleListUp := FALSE;
	IF(udiMinModuleList + 4 <= vpq_stMachineInterface.iq_stExt.udiNumberOfSubModules + vpq_stMachineInterface.iq_stExt.udiNumberOfControlModules) THEN
		udiMinModuleList := udiMinModuleList + 1;
	END_IF
	xUpdateData := TRUE;
END_IF
(* Submodule level *)
IF(udiCurrentLevel >= 2) THEN (* Impossible if the main machine is selected *)
	IF vpiq_axSubModuleList[1] OR vpiq_axSubModuleList[2] OR vpiq_axSubModuleList[3] OR vpiq_axSubModuleList[4] OR vpiq_axSubModuleList[5] OR
	   vpiq_axSubControlModuleList[1] OR vpiq_axSubControlModuleList[2] OR vpiq_axSubControlModuleList[3] OR vpiq_axSubControlModuleList[4] OR vpiq_axSubControlModuleList[5] THEN
		udiCurrentLevel := 3;
		FOR udiTmp := 1 TO 5 DO
			(*select an equipment module via the buttons on level 3*)
			IF(vpiq_axSubModuleList[udiTmp]) THEN
				audiHierarchy[udiCurrentLevel] := udiTmp + udiMinSubModuleList - 1;
				vpiq_axSubModuleList[udiTmp] := FALSE;
				udiControlModuleSelectedInLevel	:= 0;
				vpq_udiActiveControlModuleNumber	:= 0;
			END_IF
			(*select a control module via the buttons on level 3*)
			IF vpiq_axSubControlModuleList[udiTmp] THEN
				audiHierarchy[udiCurrentLevel] := udiTmp + udiMinSubModuleList - 1;
				vpiq_axSubControlModuleList[udiTmp] := FALSE;
				udiControlModuleSelectedInLevel	:= udiCurrentLevel;
			END_IF
		END_FOR
		xUpdateData := TRUE;
	END_IF
	IF vpiq_xSubModuleListDown THEN
		vpiq_xSubModuleListDown := FALSE;
		IF(udiMinSubModuleList > 1) THEN
			udiMinSubModuleList := udiMinSubModuleList - 1;
		END_IF
		xUpdateData := TRUE;
	END_IF
	IF vpiq_xSubModuleListUp THEN
		vpiq_xSubModuleListUp := FALSE;
		IF(udiMinSubModuleList + 4 < udiCurrentLevel3Size + udiNumberOfControlModulesLevel2) THEN
			udiMinSubModuleList := udiMinSubModuleList + 1;
		END_IF
		xUpdateData := TRUE;
	END_IF
END_IF
END_ACTION

ACTION ModuleNavigationOut:
(* update 2d nav data *)
vpq_sNameNavUp		:= '';
vpq_sNameNavRight	:= '';
vpq_sNameNavLeft		:= '';

IF pstCurrentParent = 0 THEN
	udiCurrentLevelSize := 1;
ELSE
	udiCurrentLevelSize := pstCurrentParent^.iq_stExt.udiNumberOfSubModules;

	vpq_sNameNavUp := pstCurrentParent^.i_sModuleName;
	(*If next module is a equipment module*)
	IF (audiHierarchy[udiCurrentLevel] + 1 <= udiCurrentLevelSize) THEN
		pstTmp := pstCurrentParent^.iq_stExt.dwSubModulesItf
			+ UDINT_TO_DWORD((audiHierarchy[udiCurrentLevel] -1 + 1) * SIZEOF(vpq_stCurrentModuleStandardInterface));
		vpq_sNameNavRight := pstTmp^.i_sModuleName;
	(*If next module is a control module*)
	ELSIF audiHierarchy[udiCurrentLevel] + 1 <= udiCurrentLevelSize + pstCurrentParent^.iq_stExt.udiNumberOfControlModules THEN
		pstControlModuleInterface	:= pstCurrentParent^.iq_stExt.dwControlModulesItf + UDINT_TO_DWORD((audiHierarchy[udiCurrentLevel]-udiCurrentLevelSize) * SIZEOF(pstControlModuleInterface^));
		vpq_sNameNavRight			:= pstControlModuleInterface^.sControlModuleName;
	END_IF
	IF (audiHierarchy[udiCurrentLevel] -1 >= 1) THEN
		(*If former module is a equipment module*)
		IF audiHierarchy[udiCurrentLevel]-1 <= udiCurrentLevelSize THEN
			pstTmp := pstCurrentParent^.iq_stExt.dwSubModulesItf
				+ UDINT_TO_DWORD((audiHierarchy[udiCurrentLevel] -1 - 1) * SIZEOF(vpq_stCurrentModuleStandardInterface));
			vpq_sNameNavLeft := pstTmp^.i_sModuleName;
		(*If former module is a control module*)
		ELSE
			pstControlModuleInterface	:= pstCurrentParent^.iq_stExt.dwControlModulesItf + UDINT_TO_DWORD((audiHierarchy[udiCurrentLevel]-udiCurrentLevelSize-2) * SIZEOF(pstControlModuleInterface^));
			vpq_sNameNavLeft				:= pstControlModuleInterface^.sControlModuleName;
		END_IF
	END_IF
END_IF

xCurrentHasControlModules := pstCurrent^.iq_stExt.udiNumberOfControlModules > 0;
xCurrentHasSubModules := ((pstCurrent^.iq_stExt.udiNumberOfSubModules > 0) AND udiControlModuleSelectedInLevel = 0);
xCurrentIsNoNodeModule := (pstCurrent^.q_dwModuleType <>  UDINT_TO_DWORD(TPL.ET_ModuleType.NodeModule));
IF((xCurrentIsNoNodeModule OR xCurrentHasControlModules) AND udiControlModuleSelectedInLevel = 0) THEN
	IF(pstCurrentParent <> 0) THEN (* Security check *)
		pdwTmp := ADR(pstCurrentParent^.iq_stExt.pdwSubModulesAddItf^)
			+  UDINT_TO_DWORD((audiHierarchy[udiCurrentLevel] - 1) * SIZEOF(dwDummy));
		dwCurrentAddInterface := pdwTmp^;
	END_IF
END_IF

vpq_xEnableNavUp		:= (udiCurrentLevel - 1 >= 1);
vpq_xEnableNavDown	:= (udiCurrentLevel < c_udiMaxHierarchyLevels) AND (xCurrentHasSubModules OR xCurrentHasControlModules) AND udiControlModuleSelectedInLevel = 0 ;
vpq_xEnableNavLeft	:= (audiHierarchy[udiCurrentLevel] -1 >= 1);
vpq_xEnableNavRight	:= (audiHierarchy[udiCurrentLevel] + 1 <= udiCurrentLevelSize + udiCurrentNumberOfControlModules)AND(udiCurrentLevel >=2);

IF vpq_xEnableNavDown THEN
	(* Name of the first submodule of the current module *)
	IF xCurrentHasSubModules THEN
		pstTmp := pstCurrent^.iq_stExt.dwSubModulesItf;
		vpq_sNameNavDown := pstTmp^.i_sModuleName;
	ELSE
		pstControlModuleInterface	:= pstCurrent^.iq_stExt.dwControlModulesItf;
		vpq_sNameNavDown				:= pstControlModuleInterface^.sControlModuleName;
	END_IF

ELSE
	vpq_sNameNavDown := '';
END_IF

(* Update direct nav data *)
(* Module level *)
vpq_xDisableModuleListDown	:= NOT (udiMinModuleList > 1);
vpq_xDisableModuleListUp		:= NOT (udiMinModuleList + 5 <= vpq_stMachineInterface.iq_stExt.udiNumberOfSubModules + vpq_stMachineInterface.iq_stExt.udiNumberOfControlModules);
FOR udiTmp := 1 TO 5 DO
	vpq_axControlModuleValid[udiTmp]:=FALSE;
	audiControlModuleNumber[udiTmp]:= 0 (*-1*);
	vpq_asToolTipControlModuleList[udiTmp] := 'None';
	vpq_axDisableModuleList[udiTmp] := NOT ((udiTmp - 1 + udiMinModuleList) <= vpq_stMachineInterface.iq_stExt.udiNumberOfSubModules);
	vpq_axActiveModuleList[udiTmp] := (udiCurrentLevel >= 2) AND (audiHierarchy[2] = (udiTmp - 1 + udiMinModuleList));
	vpq_axControlModuleActive[udiTmp] := FALSE;
	(*Show button for equipment module*)
	IF(NOT vpq_axDisableModuleList[udiTmp]) THEN
		pstTmp := vpq_stMachineInterface.iq_stExt.dwSubModulesItf
			+ UDINT_TO_DWORD(((udiTmp - 1 + udiMinModuleList) - 1) * SIZEOF(vpq_stCurrentModuleStandardInterface));
		vpq_audiIdModuleList[udiTmp] := pstTmp^.i_udiModuleId;
		vpq_axIdModuleListValid[udiTmp] := TRUE;
		
		vpq_asNameModuleList[udiTmp] := pstTmp^.i_sModuleName;
	(*Show button for control module*)
	ELSE
		vpq_audiIdModuleList[udiTmp] := 0 (*-1*);
		vpq_axIdModuleListValid[udiTmp] := FALSE;
		vpq_asNameModuleList[udiTmp] := 'None';
		IF vpq_stMachineInterface.iq_stExt.udiNumberOfControlModules <> 0 AND udiTmp <= vpq_stMachineInterface.iq_stExt.udiNumberOfControlModules + vpq_stMachineInterface.iq_stExt.udiNumberOfSubModules THEN
			pstControlModuleInterface	:= vpq_stMachineInterface.iq_stExt.dwControlModulesItf + UDINT_TO_DWORD((udiTmp - vpq_stMachineInterface.iq_stExt.udiNumberOfSubModules - 1 + udiMinModuleList)-1) * SIZEOF(pstControlModuleInterface^);
			vpq_asToolTipControlModuleList[udiTmp]:= pstControlModuleInterface^.sControlModuleName;
			vpq_axControlModuleActive[udiTmp] := (udiCurrentLevel >= 2) AND (audiHierarchy[2] = (udiTmp - 1 + udiMinModuleList));
			vpq_axControlModuleValid[udiTmp]:=TRUE;
			audiControlModuleNumber[udiTmp]:= pstControlModuleInterface^.udiControlModuleNumber;
			vpq_asControlModuleButtonName[udiTmp]:= CONCAT(STR1:='Type: ',STR2:= CONCAT(STR1:= UDINT_TO_STRING(pstControlModuleInterface^.udiControlModuleType), STR2:= CONCAT(STR1:='   #: ',STR2:= UDINT_TO_STRING(pstControlModuleInterface^.udiControlModuleNumber))));
		END_IF
	END_IF
END_FOR

(* Submodule level *)
IF (udiMinSubModuleList + 4 > udiCurrentLevel3Size+udiNumberOfControlModulesLevel2) THEN
	udiMinSubModuleList := 1;
END_IF
vpq_xDisableSubModuleListDown	:= NOT (udiMinSubModuleList > 1);
vpq_xDisableSubModuleListUp		:= NOT (udiMinSubModuleList + 5 <= udiCurrentLevel3Size+udiNumberOfControlModulesLevel2)AND NOT (udiCurrentLevel = 2 AND xControlModuleSelected);
FOR udiTmp := 1 TO 5 DO
	vpq_axDisableSubModuleList[udiTmp] := NOT ((udiTmp - 1 + udiMinSubModuleList) <= udiCurrentLevel3Size);
	vpq_axActiveSubModuleList[udiTmp] := (udiCurrentLevel >= 3) AND (audiHierarchy[3] = (udiTmp - 1 + udiMinSubModuleList));
	vpq_audiIdSubModuleList[udiTmp] := 0 (*-1*);
	vpq_axIdSubModuleListValid[udiTmp] := FALSE;
	vpq_asNameSubModuleList[udiTmp] := 'None';
	vpq_axSubControlModuleValid[udiTmp]:= FALSE;
	audiSubControlModuleID[udiTmp]:= 0 (*-1*);
	vpq_asToolTipSubControlModuleList[udiTmp] := 'None';
	vpq_axSubControlModuleActive[udiTmp] := FALSE;
	(*Show button for equipment module*)
	IF(NOT vpq_axDisableSubModuleList[udiTmp]) THEN
		IF(pstCurrentFirstLevel3Module <> 0) THEN
			pstTmp := ADR(pstCurrentFirstLevel3Module^)
				+  UDINT_TO_DWORD(((udiTmp - 1 + udiMinSubModuleList) - 1) * SIZEOF(vpq_stCurrentModuleStandardInterface));
			vpq_audiIdSubModuleList[udiTmp] := pstTmp^.i_udiModuleId;
			vpq_axIdSubModuleListValid[udiTmp] := TRUE;
			
			vpq_asNameSubModuleList[udiTmp] := pstTmp^.i_sModuleName;
		END_IF
	(*Show button for control module*)
	ELSE
		IF udiCurrentLevel >= 2 AND udiControlModuleSelectedInLevel <> 2 THEN
			IF pstCurrentLevel2 <> 0 THEN
				IF pstCurrentLevel2^.iq_stExt.udiNumberOfControlModules <> 0 AND udiTmp <= pstCurrentLevel2^.iq_stExt.udiNumberOfControlModules + udiCurrentLevel3Size THEN
					pstControlModuleInterface	:= pstCurrentLevel2^.iq_stExt.dwControlModulesItf + UDINT_TO_DWORD((udiTmp - pstCurrentLevel2^.iq_stExt.udiNumberOfSubModules - 1 + udiMinSubModuleList - 1) * SIZEOF(pstControlModuleInterface^));
					vpq_asToolTipSubControlModuleList[udiTmp]:= pstControlModuleInterface^.sControlModuleName;
					vpq_asSubControlModuleButtonName[udiTmp]:= CONCAT(STR1:='Type: ',STR2:= CONCAT(STR1:= UDINT_TO_STRING(pstControlModuleInterface^.udiControlModuleType), STR2:= CONCAT(STR1:='   #: ',STR2:= UDINT_TO_STRING(pstControlModuleInterface^.udiControlModuleNumber))));
					vpq_axSubControlModuleActive[udiTmp] :=  (udiCurrentLevel >= 3) AND (audiHierarchy[3] = (udiTmp - 1 + udiMinSubModuleList));
					vpq_axSubControlModuleValid[udiTmp]:= TRUE;
					audiSubControlModuleID[udiTmp]:= pstControlModuleInterface^.udiControlModuleNumber;
				END_IF
			END_IF
		END_IF
	END_IF
END_FOR

// iEQTableIndexMin := 1;
//iEQTableIndexOld := 0;

(*Select current control module*)
FOR udiTmp := 1 TO 5 DO
	IF vpq_axControlModuleActive[udiTmp] THEN
		vpq_udiActiveControlModuleNumber:= audiControlModuleNumber[udiTmp];
	END_IF
	IF vpq_axSubControlModuleActive[udiTmp] THEN
		vpq_udiActiveControlModuleNumber:= audiSubControlModuleID[udiTmp];
	END_IF
END_FOR
END_ACTION

ACTION ModuleReaction:
stModuleReactions		:=pstCurrent^.i_stReaction;

IF vpiq_xModuleReactionUp THEN
	vpq_udiModuleReactionIndexMin := vpq_udiModuleReactionIndexMin + 1;
	vpiq_xModuleReactionUp := FALSE;
ELSIF vpiq_xModuleReactionDown THEN
	vpq_udiModuleReactionIndexMin := vpq_udiModuleReactionIndexMin - 1;
	vpiq_xModuleReactionDown := FALSE;
END_IF

IF vpq_udiModuleReactionIndexMin <> udiModuleReactionIndexOld THEN
														(*More than 10 steps ??*)
	IF (vpq_udiModuleReactionIndexMin + 9 < TPL.Gc_udiMaxNumberOfReactions) THEN
		udiModuleReactionIndexMax := vpq_udiModuleReactionIndexMin + 9;
	ELSE
		udiModuleReactionIndexMax := TPL.Gc_udiMaxNumberOfReactions;
	END_IF
														(*Additional safety check*)
	IF (vpq_udiModuleReactionIndexMin < 1) THEN
		vpq_udiModuleReactionIndexMin :=1;
		udiModuleReactionIndexMax := 10;
 	ELSIF (vpq_udiModuleReactionIndexMin > TPL.Gc_udiMaxNumberOfReactions-9)THEN
		vpq_udiModuleReactionIndexMin :=TPL.Gc_udiMaxNumberOfReactions-9;
		udiModuleReactionIndexMax := 10;
	END_IF

	udiModuleReactionIndexOld := vpq_udiModuleReactionIndexMin;
END_IF

IF TPL.Gc_udiMaxNumberOfReactions<10 THEN
	udiMaxValue := TPL.Gc_udiMaxNumberOfReactions;
ELSE
	udiMaxValue := 10;
END_IF

FOR udiCount2 := 1 TO udiMaxValue  DO
	vpq_axModuleReaction[udiCount2] := stModuleReactions.axReaction[vpq_udiModuleReactionIndexMin + udiCount2 - 1];
END_FOR
END_ACTION

ACTION ModuleVisController:
(* Begin of area for vis control fbs of different module types *)
(* SetCurrentModule(); has to be called after each special vis-controller, because it could have requested to change the current module via diSetAsCurrentModule *)

vpiq_fbAxisModuleVisController(	i_xEnable				:= vpq_xDoEnable, 
								i_pstMachineStandardItf	:= ADR(SR_MainMachine.stMachineInterface),
								i_pstCurrentStandardItf	:= pstCurrent, 
								i_dwCurrentAddItf		:= dwCurrentAddInterface, 
								i_xUpdateData			:= xUpdateForOtherFBs,
								i_udiCurrentJogTarget	:= G_udiManualModuleSelect, 
								iq_stExceptionList		:= G_stExceptionList,
								iq_stLogDataList		:= G_stLogDataList,
								q_xActive				=> , 
								q_xReady				=> , 
								q_etDiag				=> , 
								q_etDiagExt				=> , 
								q_sMsg					=> , 
								q_udiSetAsCurrentModule	=> udiSetAsCurrentModule,
								q_udiSetAsJogTarget		=> udiSetAsJogTarget);
SetCurrentModule();

(*
vpiq_fbCrankModuleVisController(
								i_xEnable:= vpq_xDoEnable, 
								i_pstMachineStandardItf:= ADR(SR_MainMachine.stMachineInterface), 
								i_pstCurrentStandardItf:= pstCurrent, 
								i_dwCurrentAddItf:= dwCurrentAddInterface, 
								i_xUpdateData:= xUpdateForOtherFBs, 
								i_udiCurrentJogTarget:= G_udiManualModuleSelect, 
								iq_stExceptionList:= G_stExceptionList, 
								iq_stLogDataList:= G_stLogDataList, 
								q_xActive=> , 
								q_xReady=> , 
								q_etDiag=> , 
								q_etDiagExt=> , 
								q_sMsg=> , 
								q_udiSetAsCurrentModule=> udiSetAsCurrentModule, 
								q_udiSetAsJogTarget=> udiSetAsJogTarget);
*)

vpiq_fbCrankModuleVisController(
								i_xEnable:= vpq_xDoEnable, 
								i_pstCurrentStandardItf:= pstCurrent, 
								i_dwCurrentAddItf:= dwCurrentAddInterface, 
								q_xActive=> , 
								q_xReady=> , 
								q_etDiag=> , 
								q_etDiagExt=> , 
								q_sMsg=> ); 
								
(* Example *)
vpiq_fbExampleLeafModuleVisController(	i_xEnable				:= vpq_xDoEnable, 
										i_pstMachineStandardItf	:= ADR(SR_MainMachine.stMachineInterface), 
										i_pstCurrentStandardItf	:= pstCurrent, 
										i_dwCurrentAddItf		:= dwCurrentAddInterface, 
										i_xUpdateData			:= xUpdateForOtherFBs, 
										i_udiCurrentJogTarget	:= G_udiManualModuleSelect, 
										iq_stExceptionList		:= G_stExceptionList,
										iq_stLogDataList		:= G_stLogDataList, 
										q_xActive				=> , 
										q_xReady				=> , 
										q_etDiag				=> , 
										q_etDiagExt				=> , 
										q_sMsg					=> , 
										q_udiSetAsCurrentModule	=> udiSetAsCurrentModule, 
										q_udiSetAsJogTarget		=> udiSetAsJogTarget);
SetCurrentModule();


(* RoboticModule *)
(*vpiq_fbRoboticModuleVisController(	i_xEnable				:= vpq_xDoEnable, 
									i_pstMachineStandardItf	:= ADR(SR_MainMachine.stMachineInterface),
									i_pstCurrentStandardItf	:= pstCurrent, 
									i_dwCurrentAddItf		:= dwCurrentAddInterface, 
									i_xUpdateData			:= xUpdateForOtherFBs,
									i_udiCurrentJogTarget	:= G_udiManualModuleSelect, 
									iq_stExceptionList		:= G_stExceptionList,
									iq_stLogDataList		:= G_stLogDataList,
									q_xActive				=> , 
									q_xReady				=> , 
									q_etDiag				=> , 
									q_etDiagExt				=> , 
									q_sMsg					=> , 
									q_udiSetAsCurrentModule	=> udiSetAsCurrentModule,
									q_udiSetAsJogTarget		=> udiSetAsJogTarget);
SetCurrentModule();*)
END_ACTION

ACTION OpModeControl:
IFB_RTOPMode(CLK:= G_xDoPrepare OR G_xDoAuto OR G_xDoManual OR G_xDoJogMachine OR G_xDoBrakeRelease );
IF G_xDoPrepare THEN
	IF g_xPrepareActive AND G_xPrepareEpas AND IFB_RTOPMode.Q THEN
		g_xPrepareActive := FALSE;
		G_xPrepareEpas:= FALSE;
	ELSIF IFB_RTOPMode.Q THEN
		g_xPrepareActive := TRUE;
		G_xPrepareEpas:= TRUE;
	END_IF
	G_xAutoEpas := FALSE;
	G_xManualEpas := FALSE;
	G_xJogMachineEpas := FALSE;
	G_xBrakeReleaseEpas := FALSE;

ELSIF G_xDoAuto THEN
	IF G_xAutoActive AND G_xAutoEpas AND IFB_RTOPMode.Q THEN
		G_xAutoActive := FALSE;
		G_xAutoEpas := FALSE;
	ELSIF IFB_RTOPMode.Q THEN
		G_xAutoActive := TRUE;
		G_xAutoEpas := TRUE;
	END_IF
	G_xManualEpas := FALSE;
	G_xJogMachineEpas := FALSE;
	G_xBrakeReleaseEpas := FALSE;
	G_xPrepareEpas:= FALSE;

